LIN {X 0,Y 518.085,Z 283.285,A -85,B 0,C 180,E1 -4909.393,E2 -4909.393} C_VEL
LIN {X 0,Y 517.096,Z 284.359,A -85,B 0,C 180,E1 -4910.032,E2 -4910.032} C_VEL
LIN {X 0,Y 517.024,Z 284.686,A -85,B 0,C 180,E1 -4910.248,E2 -4910.248} C_VEL
LIN {X 0,Y 516.962,Z 289.338,A -85,B 0,C 180,E1 -4913.331,E2 -4913.331} C_VEL
LIN {X 0,Y 516.869,Z 293.688,A -85,B 0,C 180,E1 -4916.119,E2 -4916.119} C_VEL
LIN {X 0,Y 516.72,Z 298.275,A -85,B 0,C 180,E1 -4918.968,E2 -4918.968} C_VEL
LIN {X 0,Y 516.637,Z 302.571,A -85,B 0,C 180,E1 -4921.569,E2 -4921.569} C_VEL
LIN {X 0,Y 516.583,Z 307.01,A -85,B 0,C 180,E1 -4924.193,E2 -4924.193} C_VEL
LIN {X 0,Y 516.487,Z 311.491,A -85,B 0,C 180,E1 -4926.759,E2 -4926.759} C_VEL
LIN {X 0,Y 516.42,Z 317.774,A -85,B 0,C 180,E1 -4930.317,E2 -4930.317} C_VEL
LIN {X 0,Y 516.431,Z 317.992,A -85,B 0,C 180,E1 -4930.439,E2 -4930.439} C_VEL
LIN {X 0,Y 520.62,Z 334.551,A -85,B 0,C 180,E1 -4930.933,E2 -4930.933} C_VEL
LIN {X 0,Y 520.4,Z 349.343,A -85,B 0,C 180,E1 -4931.382,E2 -4931.382} C_VEL
LIN {X 0,Y 519.913,Z 364.135,A -85,B 0,C 180,E1 -4931.989,E2 -4931.989} C_VEL
LIN {X 0,Y 519.41,Z 378.991,A -85,B 0,C 180,E1 -4932.784,E2 -4932.784} C_VEL
LIN {X 0,Y 518.883,Z 392.399,A -85,B 0,C 180,E1 -4933.678,E2 -4933.678} C_VEL
LIN {X 0,Y 518.337,Z 404.939,A -85,B 0,C 180,E1 -4934.694,E2 -4934.694} C_VEL
LIN {X 0,Y 517.847,Z 416.905,A -85,B 0,C 180,E1 -4935.861,E2 -4935.861} C_VEL
LIN {X 0,Y 517.443,Z 427.131,A -85,B 0,C 180,E1 -4937.05,E2 -4937.05} C_VEL
LIN {X 0,Y 517.039,Z 437.144,A -85,B 0,C 180,E1 -4938.435,E2 -4938.435} C_VEL
LIN {X 0,Y 516.76,Z 445.45,A -85,B 0,C 180,E1 -4939.817,E2 -4939.817} C_VEL
LIN {X 0,Y 516.543,Z 453.254,A -85,B 0,C 180,E1 -4941.393,E2 -4941.393} C_VEL
LIN {X 0,Y 516.392,Z 459.47,A -85,B 0,C 180,E1 -4942.965,E2 -4942.965} C_VEL
LIN {X 0,Y 516.374,Z 464.272,A -85,B 0,C 180,E1 -4944.533,E2 -4944.533} C_VEL
LIN {X 0,Y 516.307,Z 467.798,A -85,B 0,C 180,E1 -4946.098,E2 -4946.098} C_VEL
LIN {X 0,Y 516.259,Z 470.138,A -85,B 0,C 180,E1 -4947.66,E2 -4947.66} C_VEL
LIN {X 0,Y 516.156,Z 471.337,A -85,B 0,C 180,E1 -4949.22,E2 -4949.22} C_VEL
LIN {X 0,Y 516.157,Z 471.356,A -85,B 0,C 180,E1 -4950.78,E2 -4950.78} C_VEL
LIN {X 0,Y 516.259,Z 470.234,A -85,B 0,C 180,E1 -4952.341,E2 -4952.341} C_VEL
LIN {X 0,Y 516.308,Z 467.969,A -85,B 0,C 180,E1 -4953.903,E2 -4953.903} C_VEL
LIN {X 0,Y 516.369,Z 464.514,A -85,B 0,C 180,E1 -4955.467,E2 -4955.467} C_VEL
LIN {X 0,Y 516.393,Z 459.789,A -85,B 0,C 180,E1 -4957.036,E2 -4957.036} C_VEL
LIN {X 0,Y 516.541,Z 453.666,A -85,B 0,C 180,E1 -4958.608,E2 -4958.608} C_VEL
LIN {X 0,Y 516.758,Z 445.959,A -85,B 0,C 180,E1 -4960.184,E2 -4960.184} C_VEL
LIN {X 0,Y 516.984,Z 437.741,A -85,B 0,C 180,E1 -4961.567,E2 -4961.567} C_VEL
LIN {X 0,Y 517.4,Z 427.847,A -85,B 0,C 180,E1 -4962.951,E2 -4962.951} C_VEL
LIN {X 0,Y 517.822,Z 417.702,A -85,B 0,C 180,E1 -4964.141,E2 -4964.141} C_VEL
LIN {X 0,Y 518.293,Z 406.094,A -85,B 0,C 180,E1 -4965.289,E2 -4965.289} C_VEL
LIN {X 0,Y 518.821,Z 393.789,A -85,B 0,C 180,E1 -4966.305,E2 -4966.305} C_VEL
LIN {X 0,Y 519.335,Z 380.39,A -85,B 0,C 180,E1 -4967.219,E2 -4967.219} C_VEL
LIN {X 0,Y 519.776,Z 367.881,A -85,B 0,C 180,E1 -4967.915,E2 -4967.915} C_VEL
LIN {X 0,Y 520.298,Z 353.859,A -85,B 0,C 180,E1 -4968.535,E2 -4968.535} C_VEL
LIN {X 0,Y 520.613,Z 339.005,A -85,B 0,C 180,E1 -4969.032,E2 -4969.032} C_VEL
LIN {X 0,Y 520.524,Z 334.046,A -85,B 0,C 180,E1 -4969.173,E2 -4969.173} C_VEL
LIN {X 0,Y 516.438,Z 317.99,A -85,B 0,C 180,E1 -4969.655,E2 -4969.655} C_VEL
LIN {X 0,Y 516.488,Z 311.675,A -85,B 0,C 180,E1 -4973.242,E2 -4973.242} C_VEL
LIN {X 0,Y 516.571,Z 306.704,A -85,B 0,C 180,E1 -4976.112,E2 -4976.112} C_VEL
LIN {X 0,Y 516.696,Z 301.285,A -85,B 0,C 180,E1 -4979.318,E2 -4979.318} C_VEL
LIN {X 0,Y 516.786,Z 296.023,A -85,B 0,C 180,E1 -4982.524,E2 -4982.524} C_VEL
LIN {X 0,Y 516.89,Z 291.549,A -85,B 0,C 180,E1 -4985.333,E2 -4985.333} C_VEL
LIN {X 0,Y 516.975,Z 287.518,A -85,B 0,C 180,E1 -4987.956,E2 -4987.956} C_VEL
LIN {X 0,Y 517.036,Z 283.394,A -85,B 0,C 180,E1 -4990.727,E2 -4990.727} C_VEL
LIN {X 0,Y 516.853,Z 280.732,A -85,B 0,C 180,E1 -4992.754,E2 -4992.754} C_VEL
LIN {X 0,Y 516.922,Z 280.722,A -85,B 0,C 180,E1 -4995.01,E2 -4995.01} C_VEL
LIN {X 0,Y 516.911,Z 280.722,A -85,B 0,C 180,E1 -4998.399,E2 -4998.399} C_VEL
LIN {X 0,Y 516.881,Z 280.725,A -85,B 0,C 180,E1 -5001.284,E2 -5001.284} C_VEL
LIN {X 0,Y 516.865,Z 280.727,A -85,B 0,C 180,E1 -5004.219,E2 -5004.219} C_VEL
LIN {X 0,Y 516.892,Z 280.723,A -85,B 0,C 180,E1 -5007.053,E2 -5007.053} C_VEL
LIN {X 0,Y 516.889,Z 280.725,A -85,B 0,C 180,E1 -5009.796,E2 -5009.796} C_VEL
LIN {X 0,Y 516.894,Z 280.727,A -85,B 0,C 180,E1 -5012.465,E2 -5012.465} C_VEL
LIN {X 0,Y 516.866,Z 280.726,A -85,B 0,C 180,E1 -5015.069,E2 -5015.069} C_VEL
LIN {X 0,Y 516.866,Z 280.725,A -85,B 0,C 180,E1 -5017.621,E2 -5017.621} C_VEL
LIN {X 0,Y 516.928,Z 280.723,A -85,B 0,C 180,E1 -5020.13,E2 -5020.13} C_VEL
LIN {X 0,Y 516.926,Z 280.719,A -85,B 0,C 180,E1 -5022.596,E2 -5022.596} C_VEL
LIN {X 0,Y 516.935,Z 280.72,A -85,B 0,C 180,E1 -5025.03,E2 -5025.03} C_VEL
LIN {X 0,Y 516.962,Z 280.715,A -85,B 0,C 180,E1 -5028.234,E2 -5028.234} C_VEL
LIN {X 0,Y 516.964,Z 280.714,A -85,B 0,C 180,E1 -5031.4,E2 -5031.4} C_VEL
LIN {X 0,Y 517.02,Z 280.707,A -85,B 0,C 180,E1 -5034.54,E2 -5034.54} C_VEL
LIN {X 0,Y 517.082,Z 280.699,A -85,B 0,C 180,E1 -5037.663,E2 -5037.663} C_VEL
LIN {X 0,Y 517.083,Z 280.699,A -85,B 0,C 180,E1 -5040.779,E2 -5040.779} C_VEL
LIN {X 0,Y 517.011,Z 280.712,A -85,B 0,C 180,E1 -5043.117,E2 -5043.117} C_VEL
LIN {X 0,Y 516.983,Z 280.715,A -85,B 0,C 180,E1 -5046.243,E2 -5046.243} C_VEL
LIN {X 0,Y 516.949,Z 280.719,A -85,B 0,C 180,E1 -5049.389,E2 -5049.389} C_VEL
LIN {X 0,Y 516.948,Z 280.717,A -85,B 0,C 180,E1 -5051.807,E2 -5051.807} C_VEL
LIN {X 0,Y 516.939,Z 280.72,A -85,B 0,C 180,E1 -5055.146,E2 -5055.146} C_VEL
LIN {X 0,Y 516.921,Z 280.722,A -85,B 0,C 180,E1 -5058.222,E2 -5058.222} C_VEL
LIN {X 0,Y 516.9,Z 280.721,A -85,B 0,C 180,E1 -5060.702,E2 -5060.702} C_VEL
LIN {X 0,Y 516.899,Z 280.723,A -85,B 0,C 180,E1 -5064.072,E2 -5064.072} C_VEL
LIN {X 0,Y 516.918,Z 280.72,A -85,B 0,C 180,E1 -5066.658,E2 -5066.658} C_VEL
LIN {X 0,Y 516.904,Z 280.724,A -85,B 0,C 180,E1 -5069.523,E2 -5069.523} C_VEL
LIN {X 0,Y 516.892,Z 280.726,A -85,B 0,C 180,E1 -5072.544,E2 -5072.544} C_VEL
LIN {X 0,Y 516.859,Z 280.734,A -85,B 0,C 180,E1 -5075.329,E2 -5075.329} C_VEL
LIN {X 0,Y 516.879,Z 280.729,A -85,B 0,C 180,E1 -5077.943,E2 -5077.943} C_VEL
LIN {X 0,Y 516.879,Z 280.726,A -85,B 0,C 180,E1 -5080.742,E2 -5080.742} C_VEL
LIN {X 0,Y 516.879,Z 280.728,A -85,B 0,C 180,E1 -5083.903,E2 -5083.903} C_VEL
LIN {X 0,Y 516.957,Z 280.907,A -85,B 0,C 180,E1 -5086.643,E2 -5086.643} C_VEL
LIN {X 0,Y 517.284,Z 283.704,A -85,B 0,C 180,E1 -5088.352,E2 -5088.352} C_VEL
LIN {X 0,Y 517.265,Z 287.849,A -85,B 0,C 180,E1 -5090.755,E2 -5090.755} C_VEL
LIN {X 0,Y 517.156,Z 292.427,A -85,B 0,C 180,E1 -5093.301,E2 -5093.301} C_VEL
LIN {X 0,Y 517.023,Z 297.711,A -85,B 0,C 180,E1 -5096.13,E2 -5096.13} C_VEL
LIN {X 0,Y 516.879,Z 303.124,A -85,B 0,C 180,E1 -5098.938,E2 -5098.938} C_VEL
LIN {X 0,Y 516.74,Z 308.364,A -85,B 0,C 180,E1 -5101.574,E2 -5101.574} C_VEL
LIN {X 0,Y 516.639,Z 313.709,A -85,B 0,C 180,E1 -5104.195,E2 -5104.195} C_VEL
LIN {X 0,Y 516.54,Z 319.079,A -85,B 0,C 180,E1 -5106.761,E2 -5106.761} C_VEL
LIN {X 0,Y 516.501,Z 325.688,A -85,B 0,C 180,E1 -5109.864,E2 -5109.864} C_VEL
LIN {X 0,Y 516.49,Z 326.814,A -85,B 0,C 180,E1 -5110.387,E2 -5110.387} C_VEL
LIN {X 0,Y 520.37,Z 342.561,A -85,B 0,C 180,E1 -5110.842,E2 -5110.842} C_VEL
LIN {X 0,Y 520.646,Z 345.506,A -85,B 0,C 180,E1 -5110.929,E2 -5110.929} C_VEL
LIN {X 0,Y 520.355,Z 359.33,A -85,B 0,C 180,E1 -5111.351,E2 -5111.351} C_VEL
LIN {X 0,Y 519.86,Z 373.609,A -85,B 0,C 180,E1 -5111.935,E2 -5111.935} C_VEL
LIN {X 0,Y 519.383,Z 387.714,A -85,B 0,C 180,E1 -5112.681,E2 -5112.681} C_VEL
LIN {X 0,Y 518.869,Z 401.448,A -85,B 0,C 180,E1 -5113.586,E2 -5113.586} C_VEL
LIN {X 0,Y 518.368,Z 413.415,A -85,B 0,C 180,E1 -5114.542,E2 -5114.542} C_VEL
LIN {X 0,Y 517.873,Z 425.158,A -85,B 0,C 180,E1 -5115.66,E2 -5115.66} C_VEL
LIN {X 0,Y 517.466,Z 435.667,A -85,B 0,C 180,E1 -5116.85,E2 -5116.85} C_VEL
LIN {X 0,Y 517.013,Z 445.939,A -85,B 0,C 180,E1 -5118.235,E2 -5118.235} C_VEL
LIN {X 0,Y 516.833,Z 454.478,A -85,B 0,C 180,E1 -5119.62,E2 -5119.62} C_VEL
LIN {X 0,Y 516.588,Z 461.58,A -85,B 0,C 180,E1 -5120.999,E2 -5120.999} C_VEL
LIN {X 0,Y 516.429,Z 468.166,A -85,B 0,C 180,E1 -5122.572,E2 -5122.572} C_VEL
LIN {X 0,Y 516.378,Z 473.318,A -85,B 0,C 180,E1 -5124.141,E2 -5124.141} C_VEL
LIN {X 0,Y 516.239,Z 476.289,A -85,B 0,C 180,E1 -5125.314,E2 -5125.314} C_VEL
LIN {X 0,Y 516.271,Z 479.183,A -85,B 0,C 180,E1 -5126.878,E2 -5126.878} C_VEL
LIN {X 0,Y 516.189,Z 480.908,A -85,B 0,C 180,E1 -5128.439,E2 -5128.439} C_VEL
LIN {X 0,Y 516.151,Z 481.5,A -85,B 0,C 180,E1 -5130,E2 -5130} C_VEL
LIN {X 0,Y 516.189,Z 480.906,A -85,B 0,C 180,E1 -5131.56,E2 -5131.56} C_VEL
LIN {X 0,Y 516.271,Z 479.178,A -85,B 0,C 180,E1 -5133.121,E2 -5133.121} C_VEL
LIN {X 0,Y 516.239,Z 476.288,A -85,B 0,C 180,E1 -5134.685,E2 -5134.685} C_VEL
LIN {X 0,Y 516.375,Z 472.162,A -85,B 0,C 180,E1 -5136.25,E2 -5136.25} C_VEL
LIN {X 0,Y 516.462,Z 466.681,A -85,B 0,C 180,E1 -5137.821,E2 -5137.821} C_VEL
LIN {X 0,Y 516.637,Z 459.705,A -85,B 0,C 180,E1 -5139.395,E2 -5139.395} C_VEL
LIN {X 0,Y 516.952,Z 451.021,A -85,B 0,C 180,E1 -5140.972,E2 -5140.972} C_VEL
LIN {X 0,Y 517.225,Z 441.942,A -85,B 0,C 180,E1 -5142.337,E2 -5142.337} C_VEL
LIN {X 0,Y 517.607,Z 432.409,A -85,B 0,C 180,E1 -5143.545,E2 -5143.545} C_VEL
LIN {X 0,Y 518.096,Z 420.241,A -85,B 0,C 180,E1 -5144.835,E2 -5144.835} C_VEL
LIN {X 0,Y 518.62,Z 408.084,A -85,B 0,C 180,E1 -5145.906,E2 -5145.906} C_VEL
LIN {X 0,Y 519.074,Z 395.608,A -85,B 0,C 180,E1 -5146.822,E2 -5146.822} C_VEL
LIN {X 0,Y 519.562,Z 382.415,A -85,B 0,C 180,E1 -5147.617,E2 -5147.617} C_VEL
LIN {X 0,Y 520.124,Z 367.924,A -85,B 0,C 180,E1 -5148.312,E2 -5148.312} C_VEL
LIN {X 0,Y 520.484,Z 353.145,A -85,B 0,C 180,E1 -5148.855,E2 -5148.855} C_VEL
LIN {X 0,Y 520.53,Z 343.102,A -85,B 0,C 180,E1 -5149.14,E2 -5149.14} C_VEL
LIN {X 0,Y 516.483,Z 326.786,A -85,B 0,C 180,E1 -5149.633,E2 -5149.633} C_VEL
LIN {X 0,Y 516.53,Z 320.903,A -85,B 0,C 180,E1 -5152.393,E2 -5152.393} C_VEL
LIN {X 0,Y 516.597,Z 315.556,A -85,B 0,C 180,E1 -5154.944,E2 -5154.944} C_VEL
LIN {X 0,Y 516.713,Z 309.555,A -85,B 0,C 180,E1 -5157.861,E2 -5157.861} C_VEL
LIN {X 0,Y 516.832,Z 304.84,A -85,B 0,C 180,E1 -5160.207,E2 -5160.207} C_VEL
LIN {X 0,Y 516.947,Z 299.493,A -85,B 0,C 180,E1 -5162.942,E2 -5162.942} C_VEL
LIN {X 0,Y 517.096,Z 294.159,A -85,B 0,C 180,E1 -5165.761,E2 -5165.761} C_VEL
LIN {X 0,Y 517.254,Z 288.849,A -85,B 0,C 180,E1 -5168.682,E2 -5168.682} C_VEL
LIN {X 0,Y 517.343,Z 285.301,A -85,B 0,C 180,E1 -5170.697,E2 -5170.697} C_VEL
LIN {X 0,Y 517.061,Z 281.779,A -85,B 0,C 180,E1 -5172.812,E2 -5172.812} C_VEL
LIN {X 0,Y 516.918,Z 280.722,A -85,B 0,C 180,E1 -5173.515,E2 -5173.515} C_VEL
LIN {X 0,Y 516.876,Z 280.728,A -85,B 0,C 180,E1 -5176.106,E2 -5176.106} C_VEL
LIN {X 0,Y 516.908,Z 280.725,A -85,B 0,C 180,E1 -5178.398,E2 -5178.398} C_VEL
LIN {X 0,Y 516.877,Z 280.726,A -85,B 0,C 180,E1 -5181.284,E2 -5181.284} C_VEL
LIN {X 0,Y 516.86,Z 280.728,A -85,B 0,C 180,E1 -5184.219,E2 -5184.219} C_VEL
LIN {X 0,Y 516.89,Z 280.725,A -85,B 0,C 180,E1 -5187.053,E2 -5187.053} C_VEL
LIN {X 0,Y 516.884,Z 280.727,A -85,B 0,C 180,E1 -5189.796,E2 -5189.796} C_VEL
LIN {X 0,Y 516.914,Z 280.725,A -85,B 0,C 180,E1 -5192.467,E2 -5192.467} C_VEL
LIN {X 0,Y 516.903,Z 280.722,A -85,B 0,C 180,E1 -5195.072,E2 -5195.072} C_VEL
LIN {X 0,Y 516.861,Z 280.727,A -85,B 0,C 180,E1 -5197.621,E2 -5197.621} C_VEL
LIN {X 0,Y 516.924,Z 280.723,A -85,B 0,C 180,E1 -5200.13,E2 -5200.13} C_VEL
LIN {X 0,Y 516.92,Z 280.719,A -85,B 0,C 180,E1 -5202.596,E2 -5202.596} C_VEL
LIN {X 0,Y 516.931,Z 280.719,A -85,B 0,C 180,E1 -5205.03,E2 -5205.03} C_VEL
LIN {X 0,Y 516.956,Z 280.715,A -85,B 0,C 180,E1 -5208.234,E2 -5208.234} C_VEL
LIN {X 0,Y 516.96,Z 280.714,A -85,B 0,C 180,E1 -5211.4,E2 -5211.4} C_VEL
LIN {X 0,Y 517.017,Z 280.706,A -85,B 0,C 180,E1 -5214.54,E2 -5214.54} C_VEL
LIN {X 0,Y 517.079,Z 280.697,A -85,B 0,C 180,E1 -5217.663,E2 -5217.663} C_VEL
LIN {X 0,Y 517.08,Z 280.699,A -85,B 0,C 180,E1 -5220.779,E2 -5220.779} C_VEL
LIN {X 0,Y 517.009,Z 280.713,A -85,B 0,C 180,E1 -5223.117,E2 -5223.117} C_VEL
LIN {X 0,Y 516.979,Z 280.716,A -85,B 0,C 180,E1 -5226.244,E2 -5226.244} C_VEL
LIN {X 0,Y 516.946,Z 280.719,A -85,B 0,C 180,E1 -5229.389,E2 -5229.389} C_VEL
LIN {X 0,Y 516.943,Z 280.716,A -85,B 0,C 180,E1 -5231.807,E2 -5231.807} C_VEL
LIN {X 0,Y 516.934,Z 280.72,A -85,B 0,C 180,E1 -5235.146,E2 -5235.146} C_VEL
LIN {X 0,Y 516.918,Z 280.722,A -85,B 0,C 180,E1 -5238.223,E2 -5238.223} C_VEL
LIN {X 0,Y 516.904,Z 280.72,A -85,B 0,C 180,E1 -5240.702,E2 -5240.702} C_VEL
LIN {X 0,Y 516.904,Z 280.722,A -85,B 0,C 180,E1 -5244.072,E2 -5244.072} C_VEL
LIN {X 0,Y 516.915,Z 280.719,A -85,B 0,C 180,E1 -5246.658,E2 -5246.658} C_VEL
LIN {X 0,Y 516.903,Z 280.721,A -85,B 0,C 180,E1 -5249.524,E2 -5249.524} C_VEL
LIN {X 0,Y 516.894,Z 280.722,A -85,B 0,C 180,E1 -5252.545,E2 -5252.545} C_VEL
LIN {X 0,Y 516.856,Z 280.73,A -85,B 0,C 180,E1 -5255.33,E2 -5255.33} C_VEL
LIN {X 0,Y 516.876,Z 280.727,A -85,B 0,C 180,E1 -5257.944,E2 -5257.944} C_VEL
LIN {X 0,Y 516.879,Z 280.725,A -85,B 0,C 180,E1 -5260.742,E2 -5260.742} C_VEL
LIN {X 0,Y 516.877,Z 280.73,A -85,B 0,C 180,E1 -5262.832,E2 -5262.832} C_VEL
LIN {X 0,Y 516.918,Z 280.72,A -85,B 0,C 180,E1 -5265.011,E2 -5265.011} C_VEL
LIN {X 0,Y 516.851,Z 280.732,A -85,B 0,C 180,E1 -5267.246,E2 -5267.246} C_VEL
LIN {X 0,Y 516.99,Z 281.991,A -85,B 0,C 180,E1 -5268.389,E2 -5268.389} C_VEL
LIN {X 0,Y 517.024,Z 284.686,A -85,B 0,C 180,E1 -5270.248,E2 -5270.248} C_VEL
LIN {X 0,Y 516.373,Z 285.721,A -85,B 0,C 180,E1 -5270.888,E2 -5270.888} C_VEL
LIN {X 0,Y 513.494,Z 287.66,A -85,B 0,C 180,E1 -5271.92,E2 -5271.92} C_VEL
LIN {X 0,Y 511.04,Z 289.243,A -85,B 0,C 180,E1 -5272.751,E2 -5272.751} C_VEL
LIN {X 0,Y 509.979,Z 290.355,A -85,B 0,C 180,E1 -5273.395,E2 -5273.395} C_VEL
LIN {X 0,Y 509.89,Z 290.698,A -85,B 0,C 180,E1 -5273.614,E2 -5273.614} C_VEL
LIN {X 0,Y 509.782,Z 295.211,A -85,B 0,C 180,E1 -5276.534,E2 -5276.534} C_VEL
LIN {X 0,Y 509.645,Z 299.658,A -85,B 0,C 180,E1 -5279.322,E2 -5279.322} C_VEL
LIN {X 0,Y 509.591,Z 304.098,A -85,B 0,C 180,E1 -5282.037,E2 -5282.037} C_VEL
LIN {X 0,Y 509.485,Z 308.546,A -85,B 0,C 180,E1 -5284.684,E2 -5284.684} C_VEL
LIN {X 0,Y 509.378,Z 313.561,A -85,B 0,C 180,E1 -5287.58,E2 -5287.58} C_VEL
LIN {X 0,Y 509.369,Z 318.129,A -85,B 0,C 180,E1 -5290.159,E2 -5290.159} C_VEL
LIN {X 0,Y 513.592,Z 334.488,A -85,B 0,C 180,E1 -5290.658,E2 -5290.658} C_VEL
LIN {X 0,Y 513.933,Z 338.016,A -85,B 0,C 180,E1 -5290.771,E2 -5290.771} C_VEL
LIN {X 0,Y 513.555,Z 353.574,A -85,B 0,C 180,E1 -5291.289,E2 -5291.289} C_VEL
LIN {X 0,Y 512.971,Z 368.2,A -85,B 0,C 180,E1 -5291.943,E2 -5291.943} C_VEL
LIN {X 0,Y 512.443,Z 382.231,A -85,B 0,C 180,E1 -5292.748,E2 -5292.748} C_VEL
LIN {X 0,Y 511.923,Z 395.059,A -85,B 0,C 180,E1 -5293.655,E2 -5293.655} C_VEL
LIN {X 0,Y 511.331,Z 407.169,A -85,B 0,C 180,E1 -5294.684,E2 -5294.684} C_VEL
LIN {X 0,Y 510.83,Z 418.764,A -85,B 0,C 180,E1 -5295.866,E2 -5295.866} C_VEL
LIN {X 0,Y 510.39,Z 428.745,A -85,B 0,C 180,E1 -5297.071,E2 -5297.071} C_VEL
LIN {X 0,Y 510,Z 438.702,A -85,B 0,C 180,E1 -5298.508,E2 -5298.508} C_VEL
LIN {X 0,Y 509.7,Z 446.621,A -85,B 0,C 180,E1 -5299.875,E2 -5299.875} C_VEL
LIN {X 0,Y 509.487,Z 453.326,A -85,B 0,C 180,E1 -5301.273,E2 -5301.273} C_VEL
LIN {X 0,Y 509.319,Z 459.541,A -85,B 0,C 180,E1 -5302.866,E2 -5302.866} C_VEL
LIN {X 0,Y 509.305,Z 464.343,A -85,B 0,C 180,E1 -5304.457,E2 -5304.457} C_VEL
LIN {X 0,Y 509.202,Z 467.865,A -85,B 0,C 180,E1 -5306.043,E2 -5306.043} C_VEL
LIN {X 0,Y 509.187,Z 470.197,A -85,B 0,C 180,E1 -5307.627,E2 -5307.627} C_VEL
LIN {X 0,Y 509.07,Z 471.393,A -85,B 0,C 180,E1 -5309.209,E2 -5309.209} C_VEL
LIN {X 0,Y 509.071,Z 471.412,A -85,B 0,C 180,E1 -5310.791,E2 -5310.791} C_VEL
LIN {X 0,Y 509.188,Z 470.291,A -85,B 0,C 180,E1 -5312.373,E2 -5312.373} C_VEL
LIN {X 0,Y 509.202,Z 468.033,A -85,B 0,C 180,E1 -5313.957,E2 -5313.957} C_VEL
LIN {X 0,Y 509.299,Z 464.581,A -85,B 0,C 180,E1 -5315.543,E2 -5315.543} C_VEL
LIN {X 0,Y 509.319,Z 459.856,A -85,B 0,C 180,E1 -5317.134,E2 -5317.134} C_VEL
LIN {X 0,Y 509.485,Z 453.733,A -85,B 0,C 180,E1 -5318.728,E2 -5318.728} C_VEL
LIN {X 0,Y 509.747,Z 446.025,A -85,B 0,C 180,E1 -5320.325,E2 -5320.325} C_VEL
LIN {X 0,Y 510.01,Z 437.485,A -85,B 0,C 180,E1 -5321.777,E2 -5321.777} C_VEL
LIN {X 0,Y 510.415,Z 427.912,A -85,B 0,C 180,E1 -5323.132,E2 -5323.132} C_VEL
LIN {X 0,Y 510.879,Z 417.766,A -85,B 0,C 180,E1 -5324.337,E2 -5324.337} C_VEL
LIN {X 0,Y 511.394,Z 406.478,A -85,B 0,C 180,E1 -5325.469,E2 -5325.469} C_VEL
LIN {X 0,Y 511.987,Z 393.592,A -85,B 0,C 180,E1 -5326.549,E2 -5326.549} C_VEL
LIN {X 0,Y 512.545,Z 380.449,A -85,B 0,C 180,E1 -5327.455,E2 -5327.455} C_VEL
LIN {X 0,Y 513.008,Z 367.937,A -85,B 0,C 180,E1 -5328.16,E2 -5328.16} C_VEL
LIN {X 0,Y 513.55,Z 354.34,A -85,B 0,C 180,E1 -5328.77,E2 -5328.77} C_VEL
LIN {X 0,Y 513.89,Z 339.691,A -85,B 0,C 180,E1 -5329.273,E2 -5329.273} C_VEL
LIN {X 0,Y 513.789,Z 335.166,A -85,B 0,C 180,E1 -5329.405,E2 -5329.405} C_VEL
LIN {X 0,Y 509.755,Z 320.075,A -85,B 0,C 180,E1 -5329.883,E2 -5329.883} C_VEL
LIN {X 0,Y 509.368,Z 318.036,A -85,B 0,C 180,E1 -5329.955,E2 -5329.955} C_VEL
LIN {X 0,Y 509.419,Z 311.73,A -85,B 0,C 180,E1 -5333.584,E2 -5333.584} C_VEL
LIN {X 0,Y 509.505,Z 307.119,A -85,B 0,C 180,E1 -5336.286,E2 -5336.286} C_VEL
LIN {X 0,Y 509.596,Z 302.818,A -85,B 0,C 180,E1 -5338.861,E2 -5338.861} C_VEL
LIN {X 0,Y 509.679,Z 298.356,A -85,B 0,C 180,E1 -5341.6,E2 -5341.6} C_VEL
LIN {X 0,Y 509.837,Z 293.877,A -85,B 0,C 180,E1 -5344.414,E2 -5344.414} C_VEL
LIN {X 0,Y 509.945,Z 289.406,A -85,B 0,C 180,E1 -5347.329,E2 -5347.329} C_VEL
LIN {X 0,Y 510.016,Z 284.924,A -85,B 0,C 180,E1 -5350.365,E2 -5350.365} C_VEL
LIN {X 0,Y 509.843,Z 281.923,A -85,B 0,C 180,E1 -5352.488,E2 -5352.488} C_VEL
LIN {X 0,Y 509.808,Z 281.608,A -85,B 0,C 180,E1 -5353.573,E2 -5353.573} C_VEL
LIN {X 0,Y 509.817,Z 281.606,A -85,B 0,C 180,E1 -5356.428,E2 -5356.428} C_VEL
LIN {X 0,Y 509.836,Z 281.602,A -85,B 0,C 180,E1 -5359.302,E2 -5359.302} C_VEL
LIN {X 0,Y 509.85,Z 281.606,A -85,B 0,C 180,E1 -5361.786,E2 -5361.786} C_VEL
LIN {X 0,Y 509.824,Z 281.607,A -85,B 0,C 180,E1 -5364.621,E2 -5364.621} C_VEL
LIN {X 0,Y 509.859,Z 281.6,A -85,B 0,C 180,E1 -5367.481,E2 -5367.481} C_VEL
LIN {X 0,Y 509.856,Z 281.599,A -85,B 0,C 180,E1 -5370.273,E2 -5370.273} C_VEL
LIN {X 0,Y 509.876,Z 281.597,A -85,B 0,C 180,E1 -5373.629,E2 -5373.629} C_VEL
LIN {X 0,Y 509.827,Z 281.603,A -85,B 0,C 180,E1 -5376.436,E2 -5376.436} C_VEL
LIN {X 0,Y 509.911,Z 281.594,A -85,B 0,C 180,E1 -5379.844,E2 -5379.844} C_VEL
LIN {X 0,Y 509.88,Z 281.6,A -85,B 0,C 180,E1 -5383.175,E2 -5383.175} C_VEL
LIN {X 0,Y 509.851,Z 281.6,A -85,B 0,C 180,E1 -5385.634,E2 -5385.634} C_VEL
LIN {X 0,Y 509.91,Z 281.593,A -85,B 0,C 180,E1 -5388.874,E2 -5388.874} C_VEL
LIN {X 0,Y 509.916,Z 281.593,A -85,B 0,C 180,E1 -5392.078,E2 -5392.078} C_VEL
LIN {X 0,Y 509.97,Z 281.585,A -85,B 0,C 180,E1 -5394.464,E2 -5394.464} C_VEL
LIN {X 0,Y 510.053,Z 281.574,A -85,B 0,C 180,E1 -5397.631,E2 -5397.631} C_VEL
LIN {X 0,Y 510.052,Z 281.579,A -85,B 0,C 180,E1 -5400,E2 -5400} C_VEL
LIN {X 0,Y 510.053,Z 281.575,A -85,B 0,C 180,E1 -5402.369,E2 -5402.369} C_VEL
LIN {X 0,Y 509.971,Z 281.585,A -85,B 0,C 180,E1 -5405.536,E2 -5405.536} C_VEL
LIN {X 0,Y 509.91,Z 281.593,A -85,B 0,C 180,E1 -5408.72,E2 -5408.72} C_VEL
LIN {X 0,Y 509.9,Z 281.595,A -85,B 0,C 180,E1 -5411.932,E2 -5411.932} C_VEL
LIN {X 0,Y 509.89,Z 281.599,A -85,B 0,C 180,E1 -5415.242,E2 -5415.242} C_VEL
LIN {X 0,Y 509.885,Z 281.597,A -85,B 0,C 180,E1 -5418.001,E2 -5418.001} C_VEL
LIN {X 0,Y 509.842,Z 281.602,A -85,B 0,C 180,E1 -5421.002,E2 -5421.002} C_VEL
LIN {X 0,Y 509.861,Z 281.603,A -85,B 0,C 180,E1 -5424.426,E2 -5424.426} C_VEL
LIN {X 0,Y 509.877,Z 281.598,A -85,B 0,C 180,E1 -5427.056,E2 -5427.056} C_VEL
LIN {X 0,Y 509.853,Z 281.601,A -85,B 0,C 180,E1 -5429.751,E2 -5429.751} C_VEL
LIN {X 0,Y 509.87,Z 281.6,A -85,B 0,C 180,E1 -5432.774,E2 -5432.774} C_VEL
LIN {X 0,Y 509.819,Z 281.608,A -85,B 0,C 180,E1 -5435.578,E2 -5435.578} C_VEL
LIN {X 0,Y 509.848,Z 281.607,A -85,B 0,C 180,E1 -5438.338,E2 -5438.338} C_VEL
LIN {X 0,Y 509.849,Z 281.605,A -85,B 0,C 180,E1 -5441.426,E2 -5441.426} C_VEL
LIN {X 0,Y 509.855,Z 281.606,A -85,B 0,C 180,E1 -5444.668,E2 -5444.668} C_VEL
LIN {X 0,Y 509.884,Z 281.764,A -85,B 0,C 180,E1 -5446.436,E2 -5446.436} C_VEL
LIN {X 0,Y 510.297,Z 285.291,A -85,B 0,C 180,E1 -5448.619,E2 -5448.619} C_VEL
LIN {X 0,Y 510.247,Z 288.818,A -85,B 0,C 180,E1 -5450.685,E2 -5450.685} C_VEL
LIN {X 0,Y 510.113,Z 294.124,A -85,B 0,C 180,E1 -5453.671,E2 -5453.671} C_VEL
LIN {X 0,Y 509.94,Z 299.443,A -85,B 0,C 180,E1 -5456.545,E2 -5456.545} C_VEL
LIN {X 0,Y 509.812,Z 304.758,A -85,B 0,C 180,E1 -5459.332,E2 -5459.332} C_VEL
LIN {X 0,Y 509.657,Z 310.091,A -85,B 0,C 180,E1 -5462.041,E2 -5462.041} C_VEL
LIN {X 0,Y 509.535,Z 315.431,A -85,B 0,C 180,E1 -5464.686,E2 -5464.686} C_VEL
LIN {X 0,Y 509.458,Z 321.376,A -85,B 0,C 180,E1 -5467.558,E2 -5467.558} C_VEL
LIN {X 0,Y 509.409,Z 326.722,A -85,B 0,C 180,E1 -5470.094,E2 -5470.094} C_VEL
LIN {X 0,Y 513.775,Z 344.464,A -85,B 0,C 180,E1 -5470.636,E2 -5470.636} C_VEL
LIN {X 0,Y 513.603,Z 359.417,A -85,B 0,C 180,E1 -5471.103,E2 -5471.103} C_VEL
LIN {X 0,Y 513.095,Z 373.54,A -85,B 0,C 180,E1 -5471.689,E2 -5471.689} C_VEL
LIN {X 0,Y 512.57,Z 387.645,A -85,B 0,C 180,E1 -5472.443,E2 -5472.443} C_VEL
LIN {X 0,Y 512.019,Z 401.238,A -85,B 0,C 180,E1 -5473.35,E2 -5473.35} C_VEL
LIN {X 0,Y 511.451,Z 413.94,A -85,B 0,C 180,E1 -5474.38,E2 -5474.38} C_VEL
LIN {X 0,Y 510.942,Z 425.088,A -85,B 0,C 180,E1 -5475.462,E2 -5475.462} C_VEL
LIN {X 0,Y 510.487,Z 435.598,A -85,B 0,C 180,E1 -5476.667,E2 -5476.667} C_VEL
LIN {X 0,Y 510.09,Z 444.513,A -85,B 0,C 180,E1 -5477.871,E2 -5477.871} C_VEL
LIN {X 0,Y 509.83,Z 453.289,A -85,B 0,C 180,E1 -5479.275,E2 -5479.275} C_VEL
LIN {X 0,Y 509.556,Z 459.639,A -85,B 0,C 180,E1 -5480.473,E2 -5480.473} C_VEL
LIN {X 0,Y 509.385,Z 466.609,A -85,B 0,C 180,E1 -5482.069,E2 -5482.069} C_VEL
LIN {X 0,Y 509.266,Z 472.087,A -85,B 0,C 180,E1 -5483.661,E2 -5483.661} C_VEL
LIN {X 0,Y 509.159,Z 476.227,A -85,B 0,C 180,E1 -5485.249,E2 -5485.249} C_VEL
LIN {X 0,Y 509.188,Z 479.13,A -85,B 0,C 180,E1 -5486.835,E2 -5486.835} C_VEL
LIN {X 0,Y 509.11,Z 480.861,A -85,B 0,C 180,E1 -5488.418,E2 -5488.418} C_VEL
LIN {X 0,Y 509.062,Z 481.454,A -85,B 0,C 180,E1 -5490,E2 -5490} C_VEL
LIN {X 0,Y 509.11,Z 480.859,A -85,B 0,C 180,E1 -5491.582,E2 -5491.582} C_VEL
LIN {X 0,Y 509.188,Z 479.126,A -85,B 0,C 180,E1 -5493.165,E2 -5493.165} C_VEL
LIN {X 0,Y 509.159,Z 476.226,A -85,B 0,C 180,E1 -5494.75,E2 -5494.75} C_VEL
LIN {X 0,Y 509.305,Z 472.093,A -85,B 0,C 180,E1 -5496.338,E2 -5496.338} C_VEL
LIN {X 0,Y 509.384,Z 466.612,A -85,B 0,C 180,E1 -5497.93,E2 -5497.93} C_VEL
LIN {X 0,Y 509.555,Z 459.635,A -85,B 0,C 180,E1 -5499.526,E2 -5499.526} C_VEL
LIN {X 0,Y 509.882,Z 452.168,A -85,B 0,C 180,E1 -5500.925,E2 -5500.925} C_VEL
LIN {X 0,Y 510.143,Z 443.433,A -85,B 0,C 180,E1 -5502.289,E2 -5502.289} C_VEL
LIN {X 0,Y 510.584,Z 433.972,A -85,B 0,C 180,E1 -5503.532,E2 -5503.532} C_VEL
LIN {X 0,Y 511.034,Z 423.143,A -85,B 0,C 180,E1 -5504.739,E2 -5504.739} C_VEL
LIN {X 0,Y 511.569,Z 411.474,A -85,B 0,C 180,E1 -5505.832,E2 -5505.832} C_VEL
LIN {X 0,Y 512.089,Z 398.395,A -85,B 0,C 180,E1 -5506.853,E2 -5506.853} C_VEL
LIN {X 0,Y 512.695,Z 384.113,A -85,B 0,C 180,E1 -5507.758,E2 -5507.758} C_VEL
LIN {X 0,Y 513.315,Z 369.506,A -85,B 0,C 180,E1 -5508.488,E2 -5508.488} C_VEL
LIN {X 0,Y 513.726,Z 354.274,A -85,B 0,C 180,E1 -5509.071,E2 -5509.071} C_VEL
LIN {X 0,Y 513.79,Z 344.288,A -85,B 0,C 180,E1 -5509.369,E2 -5509.369} C_VEL
LIN {X 0,Y 509.617,Z 328.121,A -85,B 0,C 180,E1 -5509.866,E2 -5509.866} C_VEL
LIN {X 0,Y 509.407,Z 326.717,A -85,B 0,C 180,E1 -5509.915,E2 -5509.915} C_VEL
LIN {X 0,Y 509.448,Z 320.829,A -85,B 0,C 180,E1 -5512.722,E2 -5512.722} C_VEL
LIN {X 0,Y 509.535,Z 315.492,A -85,B 0,C 180,E1 -5515.313,E2 -5515.313} C_VEL
LIN {X 0,Y 509.663,Z 309.964,A -85,B 0,C 180,E1 -5518.051,E2 -5518.051} C_VEL
LIN {X 0,Y 509.813,Z 304.797,A -85,B 0,C 180,E1 -5520.667,E2 -5520.667} C_VEL
LIN {X 0,Y 509.937,Z 299.451,A -85,B 0,C 180,E1 -5523.454,E2 -5523.454} C_VEL
LIN {X 0,Y 510.109,Z 294.121,A -85,B 0,C 180,E1 -5526.329,E2 -5526.329} C_VEL
LIN {X 0,Y 510.253,Z 288.437,A -85,B 0,C 180,E1 -5529.528,E2 -5529.528} C_VEL
LIN {X 0,Y 510.294,Z 285.28,A -85,B 0,C 180,E1 -5531.381,E2 -5531.381} C_VEL
LIN {X 0,Y 509.858,Z 281.599,A -85,B 0,C 180,E1 -5533.694,E2 -5533.694} C_VEL
LIN {X 0,Y 509.812,Z 281.607,A -85,B 0,C 180,E1 -5536.428,E2 -5536.428} C_VEL
LIN {X 0,Y 509.833,Z 281.603,A -85,B 0,C 180,E1 -5539.302,E2 -5539.302} C_VEL
LIN {X 0,Y 509.845,Z 281.606,A -85,B 0,C 180,E1 -5541.786,E2 -5541.786} C_VEL
LIN {X 0,Y 509.819,Z 281.609,A -85,B 0,C 180,E1 -5544.621,E2 -5544.621} C_VEL
LIN {X 0,Y 509.858,Z 281.603,A -85,B 0,C 180,E1 -5547.481,E2 -5547.481} C_VEL
LIN {X 0,Y 509.85,Z 281.602,A -85,B 0,C 180,E1 -5550.273,E2 -5550.273} C_VEL
LIN {X 0,Y 509.873,Z 281.599,A -85,B 0,C 180,E1 -5552.944,E2 -5552.944} C_VEL
LIN {X 0,Y 509.862,Z 281.603,A -85,B 0,C 180,E1 -5555.574,E2 -5555.574} C_VEL
LIN {X 0,Y 509.841,Z 281.602,A -85,B 0,C 180,E1 -5558.998,E2 -5558.998} C_VEL
LIN {X 0,Y 509.88,Z 281.597,A -85,B 0,C 180,E1 -5561.999,E2 -5561.999} C_VEL
LIN {X 0,Y 509.902,Z 281.596,A -85,B 0,C 180,E1 -5564.819,E2 -5564.819} C_VEL
LIN {X 0,Y 509.896,Z 281.595,A -85,B 0,C 180,E1 -5568.121,E2 -5568.121} C_VEL
LIN {X 0,Y 509.907,Z 281.593,A -85,B 0,C 180,E1 -5571.28,E2 -5571.28} C_VEL
LIN {X 0,Y 509.967,Z 281.584,A -85,B 0,C 180,E1 -5574.464,E2 -5574.464} C_VEL
LIN {X 0,Y 510.049,Z 281.573,A -85,B 0,C 180,E1 -5577.631,E2 -5577.631} C_VEL
LIN {X 0,Y 510.051,Z 281.575,A -85,B 0,C 180,E1 -5580.79,E2 -5580.79} C_VEL
LIN {X 0,Y 509.951,Z 281.591,A -85,B 0,C 180,E1 -5583.16,E2 -5583.16} C_VEL
LIN {X 0,Y 509.925,Z 281.593,A -85,B 0,C 180,E1 -5586.33,E2 -5586.33} C_VEL
LIN {X 0,Y 509.906,Z 281.592,A -85,B 0,C 180,E1 -5588.72,E2 -5588.72} C_VEL
LIN {X 0,Y 509.895,Z 281.595,A -85,B 0,C 180,E1 -5591.932,E2 -5591.932} C_VEL
LIN {X 0,Y 509.885,Z 281.599,A -85,B 0,C 180,E1 -5595.242,E2 -5595.242} C_VEL
LIN {X 0,Y 509.881,Z 281.596,A -85,B 0,C 180,E1 -5598.001,E2 -5598.001} C_VEL
LIN {X 0,Y 509.842,Z 281.601,A -85,B 0,C 180,E1 -5601.002,E2 -5601.002} C_VEL
LIN {X 0,Y 509.862,Z 281.603,A -85,B 0,C 180,E1 -5604.426,E2 -5604.426} C_VEL
LIN {X 0,Y 509.874,Z 281.597,A -85,B 0,C 180,E1 -5607.056,E2 -5607.056} C_VEL
LIN {X 0,Y 509.85,Z 281.598,A -85,B 0,C 180,E1 -5609.752,E2 -5609.752} C_VEL
LIN {X 0,Y 509.87,Z 281.596,A -85,B 0,C 180,E1 -5612.775,E2 -5612.775} C_VEL
LIN {X 0,Y 509.816,Z 281.605,A -85,B 0,C 180,E1 -5615.579,E2 -5615.579} C_VEL
LIN {X 0,Y 509.845,Z 281.605,A -85,B 0,C 180,E1 -5618.339,E2 -5618.339} C_VEL
LIN {X 0,Y 509.851,Z 281.605,A -85,B 0,C 180,E1 -5621.426,E2 -5621.426} C_VEL
LIN {X 0,Y 509.852,Z 281.602,A -85,B 0,C 180,E1 -5624.669,E2 -5624.669} C_VEL
LIN {X 0,Y 509.821,Z 281.79,A -85,B 0,C 180,E1 -5627.51,E2 -5627.51} C_VEL
LIN {X 0,Y 510.013,Z 284.793,A -85,B 0,C 180,E1 -5629.636,E2 -5629.636} C_VEL
LIN {X 0,Y 509.93,Z 289.873,A -85,B 0,C 180,E1 -5633.07,E2 -5633.07} C_VEL
LIN {X 0,Y 509.89,Z 290.698,A -85,B 0,C 180,E1 -5633.614,E2 -5633.614} C_VEL
LIN {X 0,Y 509.211,Z 291.771,A -85,B 0,C 180,E1 -5634.262,E2 -5634.262} C_VEL
LIN {X 0,Y 506.332,Z 293.742,A -85,B 0,C 180,E1 -5635.309,E2 -5635.309} C_VEL
LIN {X 0,Y 503.881,Z 295.346,A -85,B 0,C 180,E1 -5636.152,E2 -5636.152} C_VEL
LIN {X 0,Y 502.802,Z 296.488,A -85,B 0,C 180,E1 -5636.806,E2 -5636.806} C_VEL
LIN {X 0,Y 502.7,Z 296.844,A -85,B 0,C 180,E1 -5637.027,E2 -5637.027} C_VEL
LIN {X 0,Y 502.584,Z 301.725,A -85,B 0,C 180,E1 -5640.111,E2 -5640.111} C_VEL
LIN {X 0,Y 502.483,Z 305.627,A -85,B 0,C 180,E1 -5642.513,E2 -5642.513} C_VEL
LIN {X 0,Y 502.401,Z 310.459,A -85,B 0,C 180,E1 -5645.405,E2 -5645.405} C_VEL
LIN {X 0,Y 502.289,Z 314.564,A -85,B 0,C 180,E1 -5647.804,E2 -5647.804} C_VEL
LIN {X 0,Y 502.279,Z 318.165,A -85,B 0,C 180,E1 -5649.866,E2 -5649.866} C_VEL
LIN {X 0,Y 506.474,Z 334.07,A -85,B 0,C 180,E1 -5650.361,E2 -5650.361} C_VEL
LIN {X 0,Y 507.243,Z 337.721,A -85,B 0,C 180,E1 -5650.496,E2 -5650.496} C_VEL
LIN {X 0,Y 506.85,Z 352.87,A -85,B 0,C 180,E1 -5651,E2 -5651} C_VEL
LIN {X 0,Y 506.233,Z 368.281,A -85,B 0,C 180,E1 -5651.694,E2 -5651.694} C_VEL
LIN {X 0,Y 505.646,Z 382.31,A -85,B 0,C 180,E1 -5652.509,E2 -5652.509} C_VEL
LIN {X 0,Y 505.084,Z 395.131,A -85,B 0,C 180,E1 -5653.427,E2 -5653.427} C_VEL
LIN {X 0,Y 504.455,Z 407.386,A -85,B 0,C 180,E1 -5654.484,E2 -5654.484} C_VEL
LIN {X 0,Y 503.91,Z 418.839,A -85,B 0,C 180,E1 -5655.668,E2 -5655.668} C_VEL
LIN {X 0,Y 503.421,Z 428.82,A -85,B 0,C 180,E1 -5656.888,E2 -5656.888} C_VEL
LIN {X 0,Y 502.985,Z 437.505,A -85,B 0,C 180,E1 -5658.139,E2 -5658.139} C_VEL
LIN {X 0,Y 502.741,Z 445.596,A -85,B 0,C 180,E1 -5659.53,E2 -5659.53} C_VEL
LIN {X 0,Y 502.444,Z 453.398,A -85,B 0,C 180,E1 -5661.15,E2 -5661.15} C_VEL
LIN {X 0,Y 502.245,Z 459.613,A -85,B 0,C 180,E1 -5662.765,E2 -5662.765} C_VEL
LIN {X 0,Y 502.215,Z 464.414,A -85,B 0,C 180,E1 -5664.379,E2 -5664.379} C_VEL
LIN {X 0,Y 502.099,Z 467.936,A -85,B 0,C 180,E1 -5665.987,E2 -5665.987} C_VEL
LIN {X 0,Y 502.088,Z 470.267,A -85,B 0,C 180,E1 -5667.594,E2 -5667.594} C_VEL
LIN {X 0,Y 501.987,Z 471.462,A -85,B 0,C 180,E1 -5669.198,E2 -5669.198} C_VEL
LIN {X 0,Y 501.988,Z 471.48,A -85,B 0,C 180,E1 -5670.802,E2 -5670.802} C_VEL
LIN {X 0,Y 502.089,Z 470.36,A -85,B 0,C 180,E1 -5672.407,E2 -5672.407} C_VEL
LIN {X 0,Y 502.099,Z 468.101,A -85,B 0,C 180,E1 -5674.013,E2 -5674.013} C_VEL
LIN {X 0,Y 502.207,Z 464.649,A -85,B 0,C 180,E1 -5675.622,E2 -5675.622} C_VEL
LIN {X 0,Y 502.245,Z 459.923,A -85,B 0,C 180,E1 -5677.235,E2 -5677.235} C_VEL
LIN {X 0,Y 502.44,Z 453.799,A -85,B 0,C 180,E1 -5678.851,E2 -5678.851} C_VEL
LIN {X 0,Y 502.738,Z 446.09,A -85,B 0,C 180,E1 -5680.471,E2 -5680.471} C_VEL
LIN {X 0,Y 502.98,Z 438.092,A -85,B 0,C 180,E1 -5681.858,E2 -5681.858} C_VEL
LIN {X 0,Y 503.443,Z 427.976,A -85,B 0,C 180,E1 -5683.317,E2 -5683.317} C_VEL
LIN {X 0,Y 503.949,Z 417.83,A -85,B 0,C 180,E1 -5684.538,E2 -5684.538} C_VEL
LIN {X 0,Y 504.503,Z 406.818,A -85,B 0,C 180,E1 -5685.659,E2 -5685.659} C_VEL
LIN {X 0,Y 505.087,Z 394.942,A -85,B 0,C 180,E1 -5686.678,E2 -5686.678} C_VEL
LIN {X 0,Y 505.681,Z 382.088,A -85,B 0,C 180,E1 -5687.595,E2 -5687.595} C_VEL
LIN {X 0,Y 506.268,Z 367.994,A -85,B 0,C 180,E1 -5688.41,E2 -5688.41} C_VEL
LIN {X 0,Y 506.804,Z 353.107,A -85,B 0,C 180,E1 -5689.082,E2 -5689.082} C_VEL
LIN {X 0,Y 507.248,Z 338.037,A -85,B 0,C 180,E1 -5689.584,E2 -5689.584} C_VEL
LIN {X 0,Y 504.431,Z 326.097,A -85,B 0,C 180,E1 -5689.996,E2 -5689.996} C_VEL
LIN {X 0,Y 502.284,Z 318.147,A -85,B 0,C 180,E1 -5690.225,E2 -5690.225} C_VEL
LIN {X 0,Y 502.336,Z 313.265,A -85,B 0,C 180,E1 -5693.063,E2 -5693.063} C_VEL
LIN {X 0,Y 502.415,Z 308.816,A -85,B 0,C 180,E1 -5695.699,E2 -5695.699} C_VEL
LIN {X 0,Y 502.514,Z 304.36,A -85,B 0,C 180,E1 -5698.393,E2 -5698.393} C_VEL
LIN {X 0,Y 502.634,Z 299.392,A -85,B 0,C 180,E1 -5701.469,E2 -5701.469} C_VEL
LIN {X 0,Y 502.791,Z 294.721,A -85,B 0,C 180,E1 -5704.442,E2 -5704.442} C_VEL
LIN {X 0,Y 502.898,Z 290.54,A -85,B 0,C 180,E1 -5707.196,E2 -5707.196} C_VEL
LIN {X 0,Y 502.979,Z 286.453,A -85,B 0,C 180,E1 -5709.997,E2 -5709.997} C_VEL
LIN {X 0,Y 502.858,Z 283.347,A -85,B 0,C 180,E1 -5712.206,E2 -5712.206} C_VEL
LIN {X 0,Y 502.755,Z 282.487,A -85,B 0,C 180,E1 -5713.372,E2 -5713.372} C_VEL
LIN {X 0,Y 502.789,Z 282.485,A -85,B 0,C 180,E1 -5715.661,E2 -5715.661} C_VEL
LIN {X 0,Y 502.817,Z 282.478,A -85,B 0,C 180,E1 -5719.005,E2 -5719.005} C_VEL
LIN {X 0,Y 502.792,Z 282.483,A -85,B 0,C 180,E1 -5722.046,E2 -5722.046} C_VEL
LIN {X 0,Y 502.794,Z 282.484,A -85,B 0,C 180,E1 -5725.034,E2 -5725.034} C_VEL
LIN {X 0,Y 502.781,Z 282.485,A -85,B 0,C 180,E1 -5727.915,E2 -5727.915} C_VEL
LIN {X 0,Y 502.81,Z 282.479,A -85,B 0,C 180,E1 -5730.711,E2 -5730.711} C_VEL
LIN {X 0,Y 502.841,Z 282.472,A -85,B 0,C 180,E1 -5733.443,E2 -5733.443} C_VEL
LIN {X 0,Y 502.777,Z 282.482,A -85,B 0,C 180,E1 -5736.085,E2 -5736.085} C_VEL
LIN {X 0,Y 502.777,Z 282.485,A -85,B 0,C 180,E1 -5738.688,E2 -5738.688} C_VEL
LIN {X 0,Y 502.826,Z 282.474,A -85,B 0,C 180,E1 -5741.248,E2 -5741.248} C_VEL
LIN {X 0,Y 502.818,Z 282.475,A -85,B 0,C 180,E1 -5743.767,E2 -5743.767} C_VEL
LIN {X 0,Y 502.818,Z 282.48,A -85,B 0,C 180,E1 -5746.254,E2 -5746.254} C_VEL
LIN {X 0,Y 502.874,Z 282.469,A -85,B 0,C 180,E1 -5748.717,E2 -5748.717} C_VEL
LIN {X 0,Y 502.877,Z 282.469,A -85,B 0,C 180,E1 -5751.966,E2 -5751.966} C_VEL
LIN {X 0,Y 502.922,Z 282.464,A -85,B 0,C 180,E1 -5754.386,E2 -5754.386} C_VEL
LIN {X 0,Y 503.023,Z 282.45,A -85,B 0,C 180,E1 -5757.598,E2 -5757.598} C_VEL
LIN {X 0,Y 502.985,Z 282.455,A -85,B 0,C 180,E1 -5760.801,E2 -5760.801} C_VEL
LIN {X 0,Y 502.897,Z 282.47,A -85,B 0,C 180,E1 -5763.204,E2 -5763.204} C_VEL
LIN {X 0,Y 502.877,Z 282.47,A -85,B 0,C 180,E1 -5766.419,E2 -5766.419} C_VEL
LIN {X 0,Y 502.869,Z 282.471,A -85,B 0,C 180,E1 -5768.843,E2 -5768.843} C_VEL
LIN {X 0,Y 502.842,Z 282.476,A -85,B 0,C 180,E1 -5772.102,E2 -5772.102} C_VEL
LIN {X 0,Y 502.845,Z 282.477,A -85,B 0,C 180,E1 -5775.4,E2 -5775.4} C_VEL
LIN {X 0,Y 502.842,Z 282.475,A -85,B 0,C 180,E1 -5778.122,E2 -5778.122} C_VEL
LIN {X 0,Y 502.825,Z 282.475,A -85,B 0,C 180,E1 -5780.536,E2 -5780.536} C_VEL
LIN {X 0,Y 502.787,Z 282.484,A -85,B 0,C 180,E1 -5783.041,E2 -5783.041} C_VEL
LIN {X 0,Y 502.836,Z 282.475,A -85,B 0,C 180,E1 -5785.676,E2 -5785.676} C_VEL
LIN {X 0,Y 502.833,Z 282.475,A -85,B 0,C 180,E1 -5788.373,E2 -5788.373} C_VEL
LIN {X 0,Y 502.789,Z 282.482,A -85,B 0,C 180,E1 -5791.499,E2 -5791.499} C_VEL
LIN {X 0,Y 502.799,Z 282.484,A -85,B 0,C 180,E1 -5793.994,E2 -5793.994} C_VEL
LIN {X 0,Y 502.774,Z 282.486,A -85,B 0,C 180,E1 -5797.178,E2 -5797.178} C_VEL
LIN {X 0,Y 502.785,Z 282.484,A -85,B 0,C 180,E1 -5800.015,E2 -5800.015} C_VEL
LIN {X 0,Y 502.8,Z 282.48,A -85,B 0,C 180,E1 -5802.199,E2 -5802.199} C_VEL
LIN {X 0,Y 502.801,Z 282.486,A -85,B 0,C 180,E1 -5805.468,E2 -5805.468} C_VEL
LIN {X 0,Y 502.845,Z 282.537,A -85,B 0,C 180,E1 -5806.172,E2 -5806.172} C_VEL
LIN {X 0,Y 503.326,Z 286.949,A -85,B 0,C 180,E1 -5808.939,E2 -5808.939} C_VEL
LIN {X 0,Y 503.151,Z 292.319,A -85,B 0,C 180,E1 -5812.078,E2 -5812.078} C_VEL
LIN {X 0,Y 503.008,Z 297.635,A -85,B 0,C 180,E1 -5815.051,E2 -5815.051} C_VEL
LIN {X 0,Y 502.806,Z 302.943,A -85,B 0,C 180,E1 -5817.917,E2 -5817.917} C_VEL
LIN {X 0,Y 502.668,Z 308.261,A -85,B 0,C 180,E1 -5820.702,E2 -5820.702} C_VEL
LIN {X 0,Y 502.532,Z 313.795,A -85,B 0,C 180,E1 -5823.515,E2 -5823.515} C_VEL
LIN {X 0,Y 502.42,Z 318.938,A -85,B 0,C 180,E1 -5826.068,E2 -5826.068} C_VEL
LIN {X 0,Y 502.329,Z 324.29,A -85,B 0,C 180,E1 -5828.669,E2 -5828.669} C_VEL
LIN {X 0,Y 502.359,Z 326.638,A -85,B 0,C 180,E1 -5829.798,E2 -5829.798} C_VEL
LIN {X 0,Y 506.904,Z 345.086,A -85,B 0,C 180,E1 -5830.383,E2 -5830.383} C_VEL
LIN {X 0,Y 507.201,Z 347.753,A -85,B 0,C 180,E1 -5830.471,E2 -5830.471} C_VEL
LIN {X 0,Y 506.82,Z 360.928,A -85,B 0,C 180,E1 -5830.904,E2 -5830.904} C_VEL
LIN {X 0,Y 506.303,Z 374.492,A -85,B 0,C 180,E1 -5831.486,E2 -5831.486} C_VEL
LIN {X 0,Y 505.689,Z 389.197,A -85,B 0,C 180,E1 -5832.301,E2 -5832.301} C_VEL
LIN {X 0,Y 505.099,Z 402.501,A -85,B 0,C 180,E1 -5833.219,E2 -5833.219} C_VEL
LIN {X 0,Y 504.488,Z 415.741,A -85,B 0,C 180,E1 -5834.335,E2 -5834.335} C_VEL
LIN {X 0,Y 503.91,Z 426.928,A -85,B 0,C 180,E1 -5835.461,E2 -5835.461} C_VEL
LIN {X 0,Y 503.437,Z 437.158,A -85,B 0,C 180,E1 -5836.683,E2 -5836.683} C_VEL
LIN {X 0,Y 502.935,Z 447.54,A -85,B 0,C 180,E1 -5838.165,E2 -5838.165} C_VEL
LIN {X 0,Y 502.716,Z 455.458,A -85,B 0,C 180,E1 -5839.529,E2 -5839.529} C_VEL
LIN {X 0,Y 502.417,Z 463.253,A -85,B 0,C 180,E1 -5841.148,E2 -5841.148} C_VEL
LIN {X 0,Y 502.244,Z 469.454,A -85,B 0,C 180,E1 -5842.765,E2 -5842.765} C_VEL
LIN {X 0,Y 502.195,Z 474.249,A -85,B 0,C 180,E1 -5844.378,E2 -5844.378} C_VEL
LIN {X 0,Y 502.094,Z 477.76,A -85,B 0,C 180,E1 -5845.987,E2 -5845.987} C_VEL
LIN {X 0,Y 502.062,Z 480.07,A -85,B 0,C 180,E1 -5847.593,E2 -5847.593} C_VEL
LIN {X 0,Y 501.987,Z 481.232,A -85,B 0,C 180,E1 -5849.198,E2 -5849.198} C_VEL
LIN {X 0,Y 501.987,Z 481.231,A -85,B 0,C 180,E1 -5850.802,E2 -5850.802} C_VEL
LIN {X 0,Y 502.062,Z 480.066,A -85,B 0,C 180,E1 -5852.406,E2 -5852.406} C_VEL
LIN {X 0,Y 502.094,Z 477.756,A -85,B 0,C 180,E1 -5854.013,E2 -5854.013} C_VEL
LIN {X 0,Y 502.196,Z 474.251,A -85,B 0,C 180,E1 -5855.621,E2 -5855.621} C_VEL
LIN {X 0,Y 502.245,Z 469.46,A -85,B 0,C 180,E1 -5857.235,E2 -5857.235} C_VEL
LIN {X 0,Y 502.416,Z 463.252,A -85,B 0,C 180,E1 -5858.851,E2 -5858.851} C_VEL
LIN {X 0,Y 502.715,Z 455.455,A -85,B 0,C 180,E1 -5860.471,E2 -5860.471} C_VEL
LIN {X 0,Y 502.967,Z 447.425,A -85,B 0,C 180,E1 -5861.852,E2 -5861.852} C_VEL
LIN {X 0,Y 503.436,Z 437.163,A -85,B 0,C 180,E1 -5863.317,E2 -5863.317} C_VEL
LIN {X 0,Y 503.909,Z 426.935,A -85,B 0,C 180,E1 -5864.539,E2 -5864.539} C_VEL
LIN {X 0,Y 504.536,Z 414.407,A -85,B 0,C 180,E1 -5865.793,E2 -5865.793} C_VEL
LIN {X 0,Y 505.175,Z 401.183,A -85,B 0,C 180,E1 -5866.882,E2 -5866.882} C_VEL
LIN {X 0,Y 505.779,Z 387.577,A -85,B 0,C 180,E1 -5867.8,E2 -5867.8} C_VEL
LIN {X 0,Y 506.409,Z 373.485,A -85,B 0,C 180,E1 -5868.561,E2 -5868.561} C_VEL
LIN {X 0,Y 506.89,Z 358.822,A -85,B 0,C 180,E1 -5869.179,E2 -5869.179} C_VEL
LIN {X 0,Y 507.111,Z 345.819,A -85,B 0,C 180,E1 -5869.588,E2 -5869.588} C_VEL
LIN {X 0,Y 503.208,Z 330.403,A -85,B 0,C 180,E1 -5870.088,E2 -5870.088} C_VEL
LIN {X 0,Y 502.364,Z 326.671,A -85,B 0,C 180,E1 -5870.194,E2 -5870.194} C_VEL
LIN {X 0,Y 502.384,Z 320.76,A -85,B 0,C 180,E1 -5873.06,E2 -5873.06} C_VEL
LIN {X 0,Y 502.473,Z 315.443,A -85,B 0,C 180,E1 -5875.695,E2 -5875.695} C_VEL
LIN {X 0,Y 502.627,Z 310.101,A -85,B 0,C 180,E1 -5878.385,E2 -5878.385} C_VEL
LIN {X 0,Y 502.779,Z 304.749,A -85,B 0,C 180,E1 -5881.144,E2 -5881.144} C_VEL
LIN {X 0,Y 502.938,Z 299.411,A -85,B 0,C 180,E1 -5883.983,E2 -5883.983} C_VEL
LIN {X 0,Y 503.091,Z 294.089,A -85,B 0,C 180,E1 -5886.919,E2 -5886.919} C_VEL
LIN {X 0,Y 503.265,Z 288.779,A -85,B 0,C 180,E1 -5889.968,E2 -5889.968} C_VEL
LIN {X 0,Y 503.172,Z 285.25,A -85,B 0,C 180,E1 -5892.099,E2 -5892.099} C_VEL
LIN {X 0,Y 502.844,Z 282.472,A -85,B 0,C 180,E1 -5893.954,E2 -5893.954} C_VEL
LIN {X 0,Y 502.766,Z 282.486,A -85,B 0,C 180,E1 -5896.768,E2 -5896.768} C_VEL
LIN {X 0,Y 502.812,Z 282.48,A -85,B 0,C 180,E1 -5899.004,E2 -5899.004} C_VEL
LIN {X 0,Y 502.787,Z 282.483,A -85,B 0,C 180,E1 -5902.046,E2 -5902.046} C_VEL
LIN {X 0,Y 502.789,Z 282.484,A -85,B 0,C 180,E1 -5905.033,E2 -5905.033} C_VEL
LIN {X 0,Y 502.78,Z 282.487,A -85,B 0,C 180,E1 -5907.915,E2 -5907.915} C_VEL
LIN {X 0,Y 502.814,Z 282.481,A -85,B 0,C 180,E1 -5910.712,E2 -5910.712} C_VEL
LIN {X 0,Y 502.854,Z 282.473,A -85,B 0,C 180,E1 -5913.439,E2 -5913.439} C_VEL
LIN {X 0,Y 502.783,Z 282.48,A -85,B 0,C 180,E1 -5916.086,E2 -5916.086} C_VEL
LIN {X 0,Y 502.775,Z 282.485,A -85,B 0,C 180,E1 -5918.689,E2 -5918.689} C_VEL
LIN {X 0,Y 502.822,Z 282.476,A -85,B 0,C 180,E1 -5921.248,E2 -5921.248} C_VEL
LIN {X 0,Y 502.813,Z 282.477,A -85,B 0,C 180,E1 -5923.767,E2 -5923.767} C_VEL
LIN {X 0,Y 502.818,Z 282.481,A -85,B 0,C 180,E1 -5926.254,E2 -5926.254} C_VEL
LIN {X 0,Y 502.874,Z 282.468,A -85,B 0,C 180,E1 -5928.717,E2 -5928.717} C_VEL
LIN {X 0,Y 502.872,Z 282.47,A -85,B 0,C 180,E1 -5931.966,E2 -5931.966} C_VEL
LIN {X 0,Y 502.919,Z 282.462,A -85,B 0,C 180,E1 -5934.386,E2 -5934.386} C_VEL
LIN {X 0,Y 503.019,Z 282.449,A -85,B 0,C 180,E1 -5937.598,E2 -5937.598} C_VEL
LIN {X 0,Y 503.001,Z 282.453,A -85,B 0,C 180,E1 -5940.801,E2 -5940.801} C_VEL
LIN {X 0,Y 502.895,Z 282.469,A -85,B 0,C 180,E1 -5943.205,E2 -5943.205} C_VEL
LIN {X 0,Y 502.873,Z 282.471,A -85,B 0,C 180,E1 -5946.42,E2 -5946.42} C_VEL
LIN {X 0,Y 502.865,Z 282.47,A -85,B 0,C 180,E1 -5948.844,E2 -5948.844} C_VEL
LIN {X 0,Y 502.837,Z 282.475,A -85,B 0,C 180,E1 -5952.102,E2 -5952.102} C_VEL
LIN {X 0,Y 502.84,Z 282.477,A -85,B 0,C 180,E1 -5955.4,E2 -5955.4} C_VEL
LIN {X 0,Y 502.838,Z 282.475,A -85,B 0,C 180,E1 -5958.123,E2 -5958.123} C_VEL
LIN {X 0,Y 502.821,Z 282.475,A -85,B 0,C 180,E1 -5960.537,E2 -5960.537} C_VEL
LIN {X 0,Y 502.786,Z 282.484,A -85,B 0,C 180,E1 -5963.041,E2 -5963.041} C_VEL
LIN {X 0,Y 502.832,Z 282.475,A -85,B 0,C 180,E1 -5965.676,E2 -5965.676} C_VEL
LIN {X 0,Y 502.829,Z 282.473,A -85,B 0,C 180,E1 -5968.373,E2 -5968.373} C_VEL
LIN {X 0,Y 502.79,Z 282.478,A -85,B 0,C 180,E1 -5971.5,E2 -5971.5} C_VEL
LIN {X 0,Y 502.796,Z 282.479,A -85,B 0,C 180,E1 -5973.995,E2 -5973.995} C_VEL
LIN {X 0,Y 502.771,Z 282.482,A -85,B 0,C 180,E1 -5977.178,E2 -5977.178} C_VEL
LIN {X 0,Y 502.783,Z 282.484,A -85,B 0,C 180,E1 -5980.016,E2 -5980.016} C_VEL
LIN {X 0,Y 502.798,Z 282.48,A -85,B 0,C 180,E1 -5982.2,E2 -5982.2} C_VEL
LIN {X 0,Y 502.796,Z 282.48,A -85,B 0,C 180,E1 -5985.469,E2 -5985.469} C_VEL
LIN {X 0,Y 502.751,Z 282.488,A -85,B 0,C 180,E1 -5986.768,E2 -5986.768} C_VEL
LIN {X 0,Y 502.859,Z 283.317,A -85,B 0,C 180,E1 -5987.868,E2 -5987.868} C_VEL
LIN {X 0,Y 502.972,Z 286.632,A -85,B 0,C 180,E1 -5990.221,E2 -5990.221} C_VEL
LIN {X 0,Y 502.888,Z 290.788,A -85,B 0,C 180,E1 -5993.064,E2 -5993.064} C_VEL
LIN {X 0,Y 502.762,Z 295.254,A -85,B 0,C 180,E1 -5996.004,E2 -5996.004} C_VEL
LIN {X 0,Y 502.7,Z 296.844,A -85,B 0,C 180,E1 -5997.027,E2 -5997.027} C_VEL
LIN {X 0,Y 501.994,Z 297.951,A -85,B 0,C 180,E1 -5997.684,E2 -5997.684} C_VEL
LIN {X 0,Y 499.115,Z 299.953,A -85,B 0,C 180,E1 -5998.745,E2 -5998.745} C_VEL
LIN {X 0,Y 496.681,Z 301.577,A -85,B 0,C 180,E1 -5999.599,E2 -5999.599} C_VEL
LIN {X 0,Y 495.605,Z 302.744,A -85,B 0,C 180,E1 -6000.261,E2 -6000.261} C_VEL
LIN {X 0,Y 495.501,Z 303.111,A -85,B 0,C 180,E1 -6000.486,E2 -6000.486} C_VEL
LIN {X 0,Y 495.401,Z 307.724,A -85,B 0,C 180,E1 -6003.348,E2 -6003.348} C_VEL
LIN {X 0,Y 495.309,Z 311.639,A -85,B 0,C 180,E1 -6005.703,E2 -6005.703} C_VEL
LIN {X 0,Y 495.191,Z 316.114,A -85,B 0,C 180,E1 -6008.346,E2 -6008.346} C_VEL
LIN {X 0,Y 495.192,Z 318.181,A -85,B 0,C 180,E1 -6009.555,E2 -6009.555} C_VEL
LIN {X 0,Y 499.774,Z 335.428,A -85,B 0,C 180,E1 -6010.123,E2 -6010.123} C_VEL
LIN {X 0,Y 500.526,Z 339.374,A -85,B 0,C 180,E1 -6010.269,E2 -6010.269} C_VEL
LIN {X 0,Y 500.097,Z 354.544,A -85,B 0,C 180,E1 -6010.799,E2 -6010.799} C_VEL
LIN {X 0,Y 499.48,Z 368.363,A -85,B 0,C 180,E1 -6011.438,E2 -6011.438} C_VEL
LIN {X 0,Y 498.86,Z 382.39,A -85,B 0,C 180,E1 -6012.263,E2 -6012.263} C_VEL
LIN {X 0,Y 498.243,Z 395.209,A -85,B 0,C 180,E1 -6013.193,E2 -6013.193} C_VEL
LIN {X 0,Y 497.573,Z 407.62,A -85,B 0,C 180,E1 -6014.279,E2 -6014.279} C_VEL
LIN {X 0,Y 496.974,Z 418.914,A -85,B 0,C 180,E1 -6015.463,E2 -6015.463} C_VEL
LIN {X 0,Y 496.462,Z 428.894,A -85,B 0,C 180,E1 -6016.701,E2 -6016.701} C_VEL
LIN {X 0,Y 495.972,Z 438.066,A -85,B 0,C 180,E1 -6018.047,E2 -6018.047} C_VEL
LIN {X 0,Y 495.736,Z 445.669,A -85,B 0,C 180,E1 -6019.38,E2 -6019.38} C_VEL
LIN {X 0,Y 495.388,Z 453.471,A -85,B 0,C 180,E1 -6021.022,E2 -6021.022} C_VEL
LIN {X 0,Y 495.171,Z 459.684,A -85,B 0,C 180,E1 -6022.662,E2 -6022.662} C_VEL
LIN {X 0,Y 495.127,Z 464.485,A -85,B 0,C 180,E1 -6024.298,E2 -6024.298} C_VEL
LIN {X 0,Y 494.998,Z 468.006,A -85,B 0,C 180,E1 -6025.93,E2 -6025.93} C_VEL
LIN {X 0,Y 494.995,Z 470.337,A -85,B 0,C 180,E1 -6027.559,E2 -6027.559} C_VEL
LIN {X 0,Y 494.907,Z 471.531,A -85,B 0,C 180,E1 -6029.187,E2 -6029.187} C_VEL
LIN {X 0,Y 494.908,Z 471.549,A -85,B 0,C 180,E1 -6030.814,E2 -6030.814} C_VEL
LIN {X 0,Y 494.995,Z 470.428,A -85,B 0,C 180,E1 -6032.441,E2 -6032.441} C_VEL
LIN {X 0,Y 494.998,Z 468.169,A -85,B 0,C 180,E1 -6034.071,E2 -6034.071} C_VEL
LIN {X 0,Y 495.116,Z 464.716,A -85,B 0,C 180,E1 -6035.703,E2 -6035.703} C_VEL
LIN {X 0,Y 495.171,Z 459.99,A -85,B 0,C 180,E1 -6037.339,E2 -6037.339} C_VEL
LIN {X 0,Y 495.383,Z 453.866,A -85,B 0,C 180,E1 -6038.978,E2 -6038.978} C_VEL
LIN {X 0,Y 495.731,Z 446.156,A -85,B 0,C 180,E1 -6040.621,E2 -6040.621} C_VEL
LIN {X 0,Y 496.031,Z 437.428,A -85,B 0,C 180,E1 -6042.143,E2 -6042.143} C_VEL
LIN {X 0,Y 496.498,Z 428.041,A -85,B 0,C 180,E1 -6043.507,E2 -6043.507} C_VEL
LIN {X 0,Y 497.037,Z 417.894,A -85,B 0,C 180,E1 -6044.745,E2 -6044.745} C_VEL
LIN {X 0,Y 497.663,Z 406.102,A -85,B 0,C 180,E1 -6045.957,E2 -6045.957} C_VEL
LIN {X 0,Y 498.311,Z 393.715,A -85,B 0,C 180,E1 -6047.017,E2 -6047.017} C_VEL
LIN {X 0,Y 498.966,Z 380.568,A -85,B 0,C 180,E1 -6047.946,E2 -6047.946} C_VEL
LIN {X 0,Y 499.541,Z 368.05,A -85,B 0,C 180,E1 -6048.667,E2 -6048.667} C_VEL
LIN {X 0,Y 500.072,Z 353.964,A -85,B 0,C 180,E1 -6049.316,E2 -6049.316} C_VEL
LIN {X 0,Y 500.456,Z 338.27,A -85,B 0,C 180,E1 -6049.855,E2 -6049.855} C_VEL
LIN {X 0,Y 496.504,Z 323.116,A -85,B 0,C 180,E1 -6050.383,E2 -6050.383} C_VEL
LIN {X 0,Y 495.198,Z 318.167,A -85,B 0,C 180,E1 -6050.552,E2 -6050.552} C_VEL
LIN {X 0,Y 495.269,Z 313.327,A -85,B 0,C 180,E1 -6053.411,E2 -6053.411} C_VEL
LIN {X 0,Y 495.36,Z 308.871,A -85,B 0,C 180,E1 -6056.092,E2 -6056.092} C_VEL
LIN {X 0,Y 495.455,Z 304.411,A -85,B 0,C 180,E1 -6058.835,E2 -6058.835} C_VEL
LIN {X 0,Y 495.593,Z 299.867,A -85,B 0,C 180,E1 -6061.695,E2 -6061.695} C_VEL
LIN {X 0,Y 495.767,Z 295.227,A -85,B 0,C 180,E1 -6064.693,E2 -6064.693} C_VEL
LIN {X 0,Y 495.845,Z 290.965,A -85,B 0,C 180,E1 -6067.551,E2 -6067.551} C_VEL
LIN {X 0,Y 495.961,Z 286.477,A -85,B 0,C 180,E1 -6070.68,E2 -6070.68} C_VEL
LIN {X 0,Y 495.728,Z 283.48,A -85,B 0,C 180,E1 -6072.882,E2 -6072.882} C_VEL
LIN {X 0,Y 495.733,Z 283.363,A -85,B 0,C 180,E1 -6075.999,E2 -6075.999} C_VEL
LIN {X 0,Y 495.765,Z 283.355,A -85,B 0,C 180,E1 -6079.3,E2 -6079.3} C_VEL
LIN {X 0,Y 495.727,Z 283.361,A -85,B 0,C 180,E1 -6082.438,E2 -6082.438} C_VEL
LIN {X 0,Y 495.774,Z 283.355,A -85,B 0,C 180,E1 -6085.456,E2 -6085.456} C_VEL
LIN {X 0,Y 495.753,Z 283.358,A -85,B 0,C 180,E1 -6088.363,E2 -6088.363} C_VEL
LIN {X 0,Y 495.752,Z 283.357,A -85,B 0,C 180,E1 -6091.514,E2 -6091.514} C_VEL
LIN {X 0,Y 495.756,Z 283.358,A -85,B 0,C 180,E1 -6093.93,E2 -6093.93} C_VEL
LIN {X 0,Y 495.758,Z 283.359,A -85,B 0,C 180,E1 -6097.139,E2 -6097.139} C_VEL
LIN {X 0,Y 495.767,Z 283.358,A -85,B 0,C 180,E1 -6100.109,E2 -6100.109} C_VEL
LIN {X 0,Y 495.783,Z 283.353,A -85,B 0,C 180,E1 -6102.681,E2 -6102.681} C_VEL
LIN {X 0,Y 495.782,Z 283.353,A -85,B 0,C 180,E1 -6105.217,E2 -6105.217} C_VEL
LIN {X 0,Y 495.848,Z 283.344,A -85,B 0,C 180,E1 -6108.555,E2 -6108.555} C_VEL
LIN {X 0,Y 495.834,Z 283.346,A -85,B 0,C 180,E1 -6111.851,E2 -6111.851} C_VEL
LIN {X 0,Y 495.837,Z 283.347,A -85,B 0,C 180,E1 -6115.121,E2 -6115.121} C_VEL
LIN {X 0,Y 495.991,Z 283.326,A -85,B 0,C 180,E1 -6117.564,E2 -6117.564} C_VEL
LIN {X 0,Y 495.937,Z 283.333,A -85,B 0,C 180,E1 -6120.812,E2 -6120.812} C_VEL
LIN {X 0,Y 495.991,Z 283.326,A -85,B 0,C 180,E1 -6122.436,E2 -6122.436} C_VEL
LIN {X 0,Y 495.877,Z 283.341,A -85,B 0,C 180,E1 -6125.694,E2 -6125.694} C_VEL
LIN {X 0,Y 495.838,Z 283.348,A -85,B 0,C 180,E1 -6128.97,E2 -6128.97} C_VEL
LIN {X 0,Y 495.824,Z 283.35,A -85,B 0,C 180,E1 -6132.035,E2 -6132.035} C_VEL
LIN {X 0,Y 495.82,Z 283.351,A -85,B 0,C 180,E1 -6135.452,E2 -6135.452} C_VEL
LIN {X 0,Y 495.803,Z 283.353,A -85,B 0,C 180,E1 -6138.247,E2 -6138.247} C_VEL
LIN {X 0,Y 495.77,Z 283.354,A -85,B 0,C 180,E1 -6140.756,E2 -6140.756} C_VEL
LIN {X 0,Y 495.744,Z 283.358,A -85,B 0,C 180,E1 -6143.387,E2 -6143.387} C_VEL
LIN {X 0,Y 495.787,Z 283.356,A -85,B 0,C 180,E1 -6146.068,E2 -6146.068} C_VEL
LIN {X 0,Y 495.765,Z 283.358,A -85,B 0,C 180,E1 -6148.815,E2 -6148.815} C_VEL
LIN {X 0,Y 495.751,Z 283.36,A -85,B 0,C 180,E1 -6151.725,E2 -6151.725} C_VEL
LIN {X 0,Y 495.764,Z 283.359,A -85,B 0,C 180,E1 -6154.694,E2 -6154.694} C_VEL
LIN {X 0,Y 495.726,Z 283.363,A -85,B 0,C 180,E1 -6157.562,E2 -6157.562} C_VEL
LIN {X 0,Y 495.756,Z 283.359,A -85,B 0,C 180,E1 -6160.047,E2 -6160.047} C_VEL
LIN {X 0,Y 495.714,Z 283.366,A -85,B 0,C 180,E1 -6162.884,E2 -6162.884} C_VEL
LIN {X 0,Y 495.797,Z 283.478,A -85,B 0,C 180,E1 -6166.006,E2 -6166.006} C_VEL
LIN {X 0,Y 496.258,Z 287.59,A -85,B 0,C 180,E1 -6168.641,E2 -6168.641} C_VEL
LIN {X 0,Y 496.179,Z 292.288,A -85,B 0,C 180,E1 -6171.448,E2 -6171.448} C_VEL
LIN {X 0,Y 495.999,Z 297.597,A -85,B 0,C 180,E1 -6174.483,E2 -6174.483} C_VEL
LIN {X 0,Y 495.803,Z 302.898,A -85,B 0,C 180,E1 -6177.408,E2 -6177.408} C_VEL
LIN {X 0,Y 495.656,Z 308.217,A -85,B 0,C 180,E1 -6180.247,E2 -6180.247} C_VEL
LIN {X 0,Y 495.48,Z 314.174,A -85,B 0,C 180,E1 -6183.33,E2 -6183.33} C_VEL
LIN {X 0,Y 495.377,Z 318.876,A -85,B 0,C 180,E1 -6185.705,E2 -6185.705} C_VEL
LIN {X 0,Y 495.277,Z 324.22,A -85,B 0,C 180,E1 -6188.35,E2 -6188.35} C_VEL
LIN {X 0,Y 495.278,Z 326.581,A -85,B 0,C 180,E1 -6189.504,E2 -6189.504} C_VEL
LIN {X 0,Y 499.722,Z 344.238,A -85,B 0,C 180,E1 -6190.066,E2 -6190.066} C_VEL
LIN {X 0,Y 500.479,Z 348.448,A -85,B 0,C 180,E1 -6190.22,E2 -6190.22} C_VEL
LIN {X 0,Y 500.102,Z 362.714,A -85,B 0,C 180,E1 -6190.713,E2 -6190.713} C_VEL
LIN {X 0,Y 499.454,Z 376.412,A -85,B 0,C 180,E1 -6191.33,E2 -6191.33} C_VEL
LIN {X 0,Y 498.825,Z 390.711,A -85,B 0,C 180,E1 -6192.155,E2 -6192.155} C_VEL
LIN {X 0,Y 498.186,Z 403.724,A -85,B 0,C 180,E1 -6193.084,E2 -6193.084} C_VEL
LIN {X 0,Y 497.57,Z 416.048,A -85,B 0,C 180,E1 -6194.148,E2 -6194.148} C_VEL
LIN {X 0,Y 496.969,Z 426.858,A -85,B 0,C 180,E1 -6195.253,E2 -6195.253} C_VEL
LIN {X 0,Y 496.476,Z 437.088,A -85,B 0,C 180,E1 -6196.493,E2 -6196.493} C_VEL
LIN {X 0,Y 495.938,Z 446.899,A -85,B 0,C 180,E1 -6197.906,E2 -6197.906} C_VEL
LIN {X 0,Y 495.678,Z 455.388,A -85,B 0,C 180,E1 -6199.378,E2 -6199.378} C_VEL
LIN {X 0,Y 495.338,Z 463.183,A -85,B 0,C 180,E1 -6201.021,E2 -6201.021} C_VEL
LIN {X 0,Y 495.165,Z 469.384,A -85,B 0,C 180,E1 -6202.661,E2 -6202.661} C_VEL
LIN {X 0,Y 495.106,Z 474.179,A -85,B 0,C 180,E1 -6204.297,E2 -6204.297} C_VEL
LIN {X 0,Y 494.991,Z 477.691,A -85,B 0,C 180,E1 -6205.929,E2 -6205.929} C_VEL
LIN {X 0,Y 494.971,Z 480.001,A -85,B 0,C 180,E1 -6207.558,E2 -6207.558} C_VEL
LIN {X 0,Y 494.907,Z 481.163,A -85,B 0,C 180,E1 -6209.186,E2 -6209.186} C_VEL
LIN {X 0,Y 494.907,Z 481.163,A -85,B 0,C 180,E1 -6210.813,E2 -6210.813} C_VEL
LIN {X 0,Y 494.97,Z 479.997,A -85,B 0,C 180,E1 -6212.441,E2 -6212.441} C_VEL
LIN {X 0,Y 494.991,Z 477.687,A -85,B 0,C 180,E1 -6214.071,E2 -6214.071} C_VEL
LIN {X 0,Y 495.11,Z 474.182,A -85,B 0,C 180,E1 -6215.702,E2 -6215.702} C_VEL
LIN {X 0,Y 495.165,Z 469.39,A -85,B 0,C 180,E1 -6217.339,E2 -6217.339} C_VEL
LIN {X 0,Y 495.338,Z 463.183,A -85,B 0,C 180,E1 -6218.978,E2 -6218.978} C_VEL
LIN {X 0,Y 495.677,Z 455.385,A -85,B 0,C 180,E1 -6220.621,E2 -6220.621} C_VEL
LIN {X 0,Y 495.986,Z 446.723,A -85,B 0,C 180,E1 -6222.12,E2 -6222.12} C_VEL
LIN {X 0,Y 496.475,Z 437.093,A -85,B 0,C 180,E1 -6223.507,E2 -6223.507} C_VEL
LIN {X 0,Y 496.976,Z 426.865,A -85,B 0,C 180,E1 -6224.746,E2 -6224.746} C_VEL
LIN {X 0,Y 497.62,Z 414.909,A -85,B 0,C 180,E1 -6225.963,E2 -6225.963} C_VEL
LIN {X 0,Y 498.279,Z 402.445,A -85,B 0,C 180,E1 -6227.017,E2 -6227.017} C_VEL
LIN {X 0,Y 498.906,Z 389.131,A -85,B 0,C 180,E1 -6227.947,E2 -6227.947} C_VEL
LIN {X 0,Y 499.608,Z 374.435,A -85,B 0,C 180,E1 -6228.77,E2 -6228.77} C_VEL
LIN {X 0,Y 500.155,Z 359.225,A -85,B 0,C 180,E1 -6229.429,E2 -6229.429} C_VEL
LIN {X 0,Y 500.37,Z 347.103,A -85,B 0,C 180,E1 -6229.824,E2 -6229.824} C_VEL
LIN {X 0,Y 496.469,Z 331.444,A -85,B 0,C 180,E1 -6230.353,E2 -6230.353} C_VEL
LIN {X 0,Y 495.251,Z 326.563,A -85,B 0,C 180,E1 -6230.513,E2 -6230.513} C_VEL
LIN {X 0,Y 495.314,Z 320.699,A -85,B 0,C 180,E1 -6233.408,E2 -6233.408} C_VEL
LIN {X 0,Y 495.425,Z 315.39,A -85,B 0,C 180,E1 -6236.088,E2 -6236.088} C_VEL
LIN {X 0,Y 495.58,Z 310.051,A -85,B 0,C 180,E1 -6238.826,E2 -6238.826} C_VEL
LIN {X 0,Y 495.758,Z 304.536,A -85,B 0,C 180,E1 -6241.726,E2 -6241.726} C_VEL
LIN {X 0,Y 495.951,Z 299.015,A -85,B 0,C 180,E1 -6244.724,E2 -6244.724} C_VEL
LIN {X 0,Y 496.102,Z 294.049,A -85,B 0,C 180,E1 -6247.528,E2 -6247.528} C_VEL
LIN {X 0,Y 496.277,Z 288.751,A -85,B 0,C 180,E1 -6250.648,E2 -6250.648} C_VEL
LIN {X 0,Y 496.042,Z 285.211,A -85,B 0,C 180,E1 -6252.848,E2 -6252.848} C_VEL
LIN {X 0,Y 495.792,Z 283.351,A -85,B 0,C 180,E1 -6254.134,E2 -6254.134} C_VEL
LIN {X 0,Y 495.731,Z 283.363,A -85,B 0,C 180,E1 -6257.492,E2 -6257.492} C_VEL
LIN {X 0,Y 495.751,Z 283.361,A -85,B 0,C 180,E1 -6260.362,E2 -6260.362} C_VEL
LIN {X 0,Y 495.72,Z 283.365,A -85,B 0,C 180,E1 -6263.455,E2 -6263.455} C_VEL
LIN {X 0,Y 495.751,Z 283.363,A -85,B 0,C 180,E1 -6266.435,E2 -6266.435} C_VEL
LIN {X 0,Y 495.745,Z 283.364,A -85,B 0,C 180,E1 -6269.312,E2 -6269.312} C_VEL
LIN {X 0,Y 495.768,Z 283.357,A -85,B 0,C 180,E1 -6272.108,E2 -6272.108} C_VEL
LIN {X 0,Y 495.781,Z 283.353,A -85,B 0,C 180,E1 -6274.832,E2 -6274.832} C_VEL
LIN {X 0,Y 495.741,Z 283.358,A -85,B 0,C 180,E1 -6277.495,E2 -6277.495} C_VEL
LIN {X 0,Y 495.764,Z 283.358,A -85,B 0,C 180,E1 -6280.109,E2 -6280.109} C_VEL
LIN {X 0,Y 495.777,Z 283.353,A -85,B 0,C 180,E1 -6282.681,E2 -6282.681} C_VEL
LIN {X 0,Y 495.779,Z 283.352,A -85,B 0,C 180,E1 -6285.217,E2 -6285.217} C_VEL
LIN {X 0,Y 495.847,Z 283.343,A -85,B 0,C 180,E1 -6288.555,E2 -6288.555} C_VEL
LIN {X 0,Y 495.829,Z 283.346,A -85,B 0,C 180,E1 -6291.851,E2 -6291.851} C_VEL
LIN {X 0,Y 495.834,Z 283.346,A -85,B 0,C 180,E1 -6295.122,E2 -6295.122} C_VEL
LIN {X 0,Y 495.987,Z 283.325,A -85,B 0,C 180,E1 -6297.564,E2 -6297.564} C_VEL
LIN {X 0,Y 495.952,Z 283.331,A -85,B 0,C 180,E1 -6300.812,E2 -6300.812} C_VEL
LIN {X 0,Y 495.987,Z 283.326,A -85,B 0,C 180,E1 -6302.436,E2 -6302.436} C_VEL
LIN {X 0,Y 495.874,Z 283.342,A -85,B 0,C 180,E1 -6305.694,E2 -6305.694} C_VEL
LIN {X 0,Y 495.834,Z 283.347,A -85,B 0,C 180,E1 -6308.97,E2 -6308.97} C_VEL
LIN {X 0,Y 495.82,Z 283.349,A -85,B 0,C 180,E1 -6312.035,E2 -6312.035} C_VEL
LIN {X 0,Y 495.815,Z 283.352,A -85,B 0,C 180,E1 -6315.452,E2 -6315.452} C_VEL
LIN {X 0,Y 495.799,Z 283.353,A -85,B 0,C 180,E1 -6318.248,E2 -6318.248} C_VEL
LIN {X 0,Y 495.766,Z 283.354,A -85,B 0,C 180,E1 -6320.757,E2 -6320.757} C_VEL
LIN {X 0,Y 495.744,Z 283.358,A -85,B 0,C 180,E1 -6323.388,E2 -6323.388} C_VEL
LIN {X 0,Y 495.784,Z 283.356,A -85,B 0,C 180,E1 -6326.068,E2 -6326.068} C_VEL
LIN {X 0,Y 495.762,Z 283.356,A -85,B 0,C 180,E1 -6328.816,E2 -6328.816} C_VEL
LIN {X 0,Y 495.752,Z 283.355,A -85,B 0,C 180,E1 -6331.727,E2 -6331.727} C_VEL
LIN {X 0,Y 495.76,Z 283.354,A -85,B 0,C 180,E1 -6334.694,E2 -6334.694} C_VEL
LIN {X 0,Y 495.723,Z 283.36,A -85,B 0,C 180,E1 -6337.562,E2 -6337.562} C_VEL
LIN {X 0,Y 495.761,Z 283.356,A -85,B 0,C 180,E1 -6340.701,E2 -6340.701} C_VEL
LIN {X 0,Y 495.729,Z 283.36,A -85,B 0,C 180,E1 -6344.002,E2 -6344.002} C_VEL
LIN {X 0,Y 495.694,Z 283.367,A -85,B 0,C 180,E1 -6347.115,E2 -6347.115} C_VEL
LIN {X 0,Y 495.958,Z 286.35,A -85,B 0,C 180,E1 -6349.32,E2 -6349.32} C_VEL
LIN {X 0,Y 495.844,Z 290.954,A -85,B 0,C 180,E1 -6352.536,E2 -6352.536} C_VEL
LIN {X 0,Y 495.752,Z 295.296,A -85,B 0,C 180,E1 -6355.456,E2 -6355.456} C_VEL
LIN {X 0,Y 495.58,Z 299.752,A -85,B 0,C 180,E1 -6358.352,E2 -6358.352} C_VEL
LIN {X 0,Y 495.501,Z 303.111,A -85,B 0,C 180,E1 -6360.486,E2 -6360.486} C_VEL
LIN {X 0,Y 494.779,Z 304.248,A -85,B 0,C 180,E1 -6361.151,E2 -6361.151} C_VEL
LIN {X 0,Y 491.873,Z 306.281,A -85,B 0,C 180,E1 -6362.227,E2 -6362.227} C_VEL
LIN {X 0,Y 489.434,Z 307.93,A -85,B 0,C 180,E1 -6363.093,E2 -6363.093} C_VEL
LIN {X 0,Y 488.377,Z 309.125,A -85,B 0,C 180,E1 -6363.764,E2 -6363.764} C_VEL
LIN {X 0,Y 488.284,Z 309.504,A -85,B 0,C 180,E1 -6363.992,E2 -6363.992} C_VEL
LIN {X 0,Y 488.218,Z 313.19,A -85,B 0,C 180,E1 -6366.231,E2 -6366.231} C_VEL
LIN {X 0,Y 488.125,Z 318.255,A -85,B 0,C 180,E1 -6369.25,E2 -6369.25} C_VEL
LIN {X 0,Y 492.616,Z 334.754,A -85,B 0,C 180,E1 -6369.798,E2 -6369.798} C_VEL
LIN {X 0,Y 493.85,Z 340.763,A -85,B 0,C 180,E1 -6370.03,E2 -6370.03} C_VEL
LIN {X 0,Y 493.382,Z 355.047,A -85,B 0,C 180,E1 -6370.544,E2 -6370.544} C_VEL
LIN {X 0,Y 492.746,Z 368.445,A -85,B 0,C 180,E1 -6371.174,E2 -6371.174} C_VEL
LIN {X 0,Y 492.095,Z 382.469,A -85,B 0,C 180,E1 -6372.011,E2 -6372.011} C_VEL
LIN {X 0,Y 491.413,Z 395.286,A -85,B 0,C 180,E1 -6372.952,E2 -6372.952} C_VEL
LIN {X 0,Y 490.696,Z 407.867,A -85,B 0,C 180,E1 -6374.07,E2 -6374.07} C_VEL
LIN {X 0,Y 490.081,Z 418.989,A -85,B 0,C 180,E1 -6375.254,E2 -6375.254} C_VEL
LIN {X 0,Y 489.516,Z 428.968,A -85,B 0,C 180,E1 -6376.509,E2 -6376.509} C_VEL
LIN {X 0,Y 488.961,Z 438.6,A -85,B 0,C 180,E1 -6377.951,E2 -6377.951} C_VEL
LIN {X 0,Y 488.638,Z 446.839,A -85,B 0,C 180,E1 -6379.434,E2 -6379.434} C_VEL
LIN {X 0,Y 488.322,Z 453.543,A -85,B 0,C 180,E1 -6380.891,E2 -6380.891} C_VEL
LIN {X 0,Y 488.122,Z 459.756,A -85,B 0,C 180,E1 -6382.555,E2 -6382.555} C_VEL
LIN {X 0,Y 488.043,Z 464.556,A -85,B 0,C 180,E1 -6384.215,E2 -6384.215} C_VEL
LIN {X 0,Y 487.899,Z 468.076,A -85,B 0,C 180,E1 -6385.87,E2 -6385.87} C_VEL
LIN {X 0,Y 487.905,Z 470.406,A -85,B 0,C 180,E1 -6387.524,E2 -6387.524} C_VEL
LIN {X 0,Y 487.83,Z 471.6,A -85,B 0,C 180,E1 -6389.175,E2 -6389.175} C_VEL
LIN {X 0,Y 487.831,Z 471.618,A -85,B 0,C 180,E1 -6390.826,E2 -6390.826} C_VEL
LIN {X 0,Y 487.906,Z 470.497,A -85,B 0,C 180,E1 -6392.477,E2 -6392.477} C_VEL
LIN {X 0,Y 487.898,Z 468.237,A -85,B 0,C 180,E1 -6394.13,E2 -6394.13} C_VEL
LIN {X 0,Y 488.028,Z 464.784,A -85,B 0,C 180,E1 -6395.786,E2 -6395.786} C_VEL
LIN {X 0,Y 488.119,Z 460.057,A -85,B 0,C 180,E1 -6397.446,E2 -6397.446} C_VEL
LIN {X 0,Y 488.313,Z 453.933,A -85,B 0,C 180,E1 -6399.109,E2 -6399.109} C_VEL
LIN {X 0,Y 488.722,Z 446.222,A -85,B 0,C 180,E1 -6400.775,E2 -6400.775} C_VEL
LIN {X 0,Y 489.023,Z 437.988,A -85,B 0,C 180,E1 -6402.241,E2 -6402.241} C_VEL
LIN {X 0,Y 489.562,Z 428.105,A -85,B 0,C 180,E1 -6403.702,E2 -6403.702} C_VEL
LIN {X 0,Y 490.108,Z 417.958,A -85,B 0,C 180,E1 -6404.958,E2 -6404.958} C_VEL
LIN {X 0,Y 490.726,Z 407.608,A -85,B 0,C 180,E1 -6406.044,E2 -6406.044} C_VEL
LIN {X 0,Y 491.417,Z 395.065,A -85,B 0,C 180,E1 -6407.156,E2 -6407.156} C_VEL
LIN {X 0,Y 492.116,Z 382.206,A -85,B 0,C 180,E1 -6408.096,E2 -6408.096} C_VEL
LIN {X 0,Y 492.703,Z 370.093,A -85,B 0,C 180,E1 -6408.828,E2 -6408.828} C_VEL
LIN {X 0,Y 493.345,Z 355.794,A -85,B 0,C 180,E1 -6409.516,E2 -6409.516} C_VEL
LIN {X 0,Y 493.796,Z 341.474,A -85,B 0,C 180,E1 -6410.041,E2 -6410.041} C_VEL
LIN {X 0,Y 493.559,Z 338.831,A -85,B 0,C 180,E1 -6410.13,E2 -6410.13} C_VEL
LIN {X 0,Y 489.853,Z 324.505,A -85,B 0,C 180,E1 -6410.648,E2 -6410.648} C_VEL
LIN {X 0,Y 488.141,Z 318.264,A -85,B 0,C 180,E1 -6410.845,E2 -6410.845} C_VEL
LIN {X 0,Y 488.217,Z 313.384,A -85,B 0,C 180,E1 -6413.77,E2 -6413.77} C_VEL
LIN {X 0,Y 488.331,Z 308.378,A -85,B 0,C 180,E1 -6416.837,E2 -6416.837} C_VEL
LIN {X 0,Y 488.439,Z 304.465,A -85,B 0,C 180,E1 -6419.289,E2 -6419.289} C_VEL
LIN {X 0,Y 488.566,Z 299.983,A -85,B 0,C 180,E1 -6422.157,E2 -6422.157} C_VEL
LIN {X 0,Y 488.727,Z 295.494,A -85,B 0,C 180,E1 -6425.114,E2 -6425.114} C_VEL
LIN {X 0,Y 488.807,Z 291.004,A -85,B 0,C 180,E1 -6428.188,E2 -6428.188} C_VEL
LIN {X 0,Y 488.948,Z 287.903,A -85,B 0,C 180,E1 -6430.376,E2 -6430.376} C_VEL
LIN {X 0,Y 488.723,Z 284.6,A -85,B 0,C 180,E1 -6432.828,E2 -6432.828} C_VEL
LIN {X 0,Y 488.694,Z 284.24,A -85,B 0,C 180,E1 -6434.023,E2 -6434.023} C_VEL
LIN {X 0,Y 488.708,Z 284.239,A -85,B 0,C 180,E1 -6437.173,E2 -6437.173} C_VEL
LIN {X 0,Y 488.732,Z 284.23,A -85,B 0,C 180,E1 -6439.676,E2 -6439.676} C_VEL
LIN {X 0,Y 488.677,Z 284.24,A -85,B 0,C 180,E1 -6442.841,E2 -6442.841} C_VEL
LIN {X 0,Y 488.727,Z 284.233,A -85,B 0,C 180,E1 -6445.887,E2 -6445.887} C_VEL
LIN {X 0,Y 488.689,Z 284.237,A -85,B 0,C 180,E1 -6448.82,E2 -6448.82} C_VEL
LIN {X 0,Y 488.709,Z 284.233,A -85,B 0,C 180,E1 -6451.669,E2 -6451.669} C_VEL
LIN {X 0,Y 488.711,Z 284.234,A -85,B 0,C 180,E1 -6454.442,E2 -6454.442} C_VEL
LIN {X 0,Y 488.721,Z 284.235,A -85,B 0,C 180,E1 -6457.153,E2 -6457.153} C_VEL
LIN {X 0,Y 488.721,Z 284.233,A -85,B 0,C 180,E1 -6459.81,E2 -6459.81} C_VEL
LIN {X 0,Y 488.73,Z 284.231,A -85,B 0,C 180,E1 -6462.423,E2 -6462.423} C_VEL
LIN {X 0,Y 488.756,Z 284.23,A -85,B 0,C 180,E1 -6464.999,E2 -6464.999} C_VEL
LIN {X 0,Y 488.802,Z 284.222,A -85,B 0,C 180,E1 -6468.387,E2 -6468.387} C_VEL
LIN {X 0,Y 488.783,Z 284.223,A -85,B 0,C 180,E1 -6471.733,E2 -6471.733} C_VEL
LIN {X 0,Y 488.833,Z 284.22,A -85,B 0,C 180,E1 -6474.224,E2 -6474.224} C_VEL
LIN {X 0,Y 488.959,Z 284.202,A -85,B 0,C 180,E1 -6477.529,E2 -6477.529} C_VEL
LIN {X 0,Y 488.964,Z 284.206,A -85,B 0,C 180,E1 -6480,E2 -6480} C_VEL
LIN {X 0,Y 488.959,Z 284.202,A -85,B 0,C 180,E1 -6482.471,E2 -6482.471} C_VEL
LIN {X 0,Y 488.834,Z 284.219,A -85,B 0,C 180,E1 -6485.776,E2 -6485.776} C_VEL
LIN {X 0,Y 488.783,Z 284.224,A -85,B 0,C 180,E1 -6488.267,E2 -6488.267} C_VEL
LIN {X 0,Y 488.802,Z 284.222,A -85,B 0,C 180,E1 -6491.612,E2 -6491.612} C_VEL
LIN {X 0,Y 488.757,Z 284.229,A -85,B 0,C 180,E1 -6495,E2 -6495} C_VEL
LIN {X 0,Y 488.752,Z 284.233,A -85,B 0,C 180,E1 -6498.442,E2 -6498.442} C_VEL
LIN {X 0,Y 488.702,Z 284.235,A -85,B 0,C 180,E1 -6501.071,E2 -6501.071} C_VEL
LIN {X 0,Y 488.685,Z 284.236,A -85,B 0,C 180,E1 -6503.746,E2 -6503.746} C_VEL
LIN {X 0,Y 488.787,Z 284.224,A -85,B 0,C 180,E1 -6506.943,E2 -6506.943} C_VEL
LIN {X 0,Y 488.705,Z 284.238,A -85,B 0,C 180,E1 -6510.363,E2 -6510.363} C_VEL
LIN {X 0,Y 488.731,Z 284.237,A -85,B 0,C 180,E1 -6513.484,E2 -6513.484} C_VEL
LIN {X 0,Y 488.678,Z 284.242,A -85,B 0,C 180,E1 -6516.354,E2 -6516.354} C_VEL
LIN {X 0,Y 488.699,Z 284.238,A -85,B 0,C 180,E1 -6519.254,E2 -6519.254} C_VEL
LIN {X 0,Y 488.685,Z 284.24,A -85,B 0,C 180,E1 -6522.526,E2 -6522.526} C_VEL
LIN {X 0,Y 488.747,Z 284.294,A -85,B 0,C 180,E1 -6525.758,E2 -6525.758} C_VEL
LIN {X 0,Y 489.226,Z 288.231,A -85,B 0,C 180,E1 -6528.332,E2 -6528.332} C_VEL
LIN {X 0,Y 489.183,Z 292.4,A -85,B 0,C 180,E1 -6530.878,E2 -6530.878} C_VEL
LIN {X 0,Y 489.006,Z 297.558,A -85,B 0,C 180,E1 -6533.896,E2 -6533.896} C_VEL
LIN {X 0,Y 488.789,Z 302.857,A -85,B 0,C 180,E1 -6536.881,E2 -6536.881} C_VEL
LIN {X 0,Y 488.643,Z 308.165,A -85,B 0,C 180,E1 -6539.775,E2 -6539.775} C_VEL
LIN {X 0,Y 488.437,Z 313.485,A -85,B 0,C 180,E1 -6542.585,E2 -6542.585} C_VEL
LIN {X 0,Y 488.347,Z 318.817,A -85,B 0,C 180,E1 -6545.333,E2 -6545.333} C_VEL
LIN {X 0,Y 488.201,Z 324.154,A -85,B 0,C 180,E1 -6548.02,E2 -6548.02} C_VEL
LIN {X 0,Y 488.174,Z 326.517,A -85,B 0,C 180,E1 -6549.194,E2 -6549.194} C_VEL
LIN {X 0,Y 492.54,Z 343.644,A -85,B 0,C 180,E1 -6549.748,E2 -6549.748} C_VEL
LIN {X 0,Y 493.75,Z 349.495,A -85,B 0,C 180,E1 -6549.972,E2 -6549.972} C_VEL
LIN {X 0,Y 493.369,Z 363.215,A -85,B 0,C 180,E1 -6550.463,E2 -6550.463} C_VEL
LIN {X 0,Y 492.72,Z 376.343,A -85,B 0,C 180,E1 -6551.065,E2 -6551.065} C_VEL
LIN {X 0,Y 492.036,Z 390.641,A -85,B 0,C 180,E1 -6551.901,E2 -6551.901} C_VEL
LIN {X 0,Y 491.352,Z 403.654,A -85,B 0,C 180,E1 -6552.842,E2 -6552.842} C_VEL
LIN {X 0,Y 490.656,Z 416.351,A -85,B 0,C 180,E1 -6553.956,E2 -6553.956} C_VEL
LIN {X 0,Y 490.037,Z 426.789,A -85,B 0,C 180,E1 -6555.039,E2 -6555.039} C_VEL
LIN {X 0,Y 489.515,Z 437.019,A -85,B 0,C 180,E1 -6556.297,E2 -6556.297} C_VEL
LIN {X 0,Y 488.899,Z 447.428,A -85,B 0,C 180,E1 -6557.825,E2 -6557.825} C_VEL
LIN {X 0,Y 488.639,Z 455.318,A -85,B 0,C 180,E1 -6559.223,E2 -6559.223} C_VEL
LIN {X 0,Y 488.274,Z 463.114,A -85,B 0,C 180,E1 -6560.89,E2 -6560.89} C_VEL
LIN {X 0,Y 488.075,Z 469.315,A -85,B 0,C 180,E1 -6562.554,E2 -6562.554} C_VEL
LIN {X 0,Y 488.001,Z 474.11,A -85,B 0,C 180,E1 -6564.214,E2 -6564.214} C_VEL
LIN {X 0,Y 487.89,Z 477.622,A -85,B 0,C 180,E1 -6565.869,E2 -6565.869} C_VEL
LIN {X 0,Y 487.883,Z 479.932,A -85,B 0,C 180,E1 -6567.523,E2 -6567.523} C_VEL
LIN {X 0,Y 487.83,Z 481.094,A -85,B 0,C 180,E1 -6569.174,E2 -6569.174} C_VEL
LIN {X 0,Y 487.83,Z 481.094,A -85,B 0,C 180,E1 -6570.825,E2 -6570.825} C_VEL
LIN {X 0,Y 487.883,Z 479.928,A -85,B 0,C 180,E1 -6572.476,E2 -6572.476} C_VEL
LIN {X 0,Y 487.89,Z 477.618,A -85,B 0,C 180,E1 -6574.13,E2 -6574.13} C_VEL
LIN {X 0,Y 488.01,Z 474.113,A -85,B 0,C 180,E1 -6575.785,E2 -6575.785} C_VEL
LIN {X 0,Y 488.075,Z 469.321,A -85,B 0,C 180,E1 -6577.446,E2 -6577.446} C_VEL
LIN {X 0,Y 488.274,Z 463.113,A -85,B 0,C 180,E1 -6579.109,E2 -6579.109} C_VEL
LIN {X 0,Y 488.636,Z 455.315,A -85,B 0,C 180,E1 -6580.776,E2 -6580.776} C_VEL
LIN {X 0,Y 488.962,Z 447.212,A -85,B 0,C 180,E1 -6582.209,E2 -6582.209} C_VEL
LIN {X 0,Y 489.515,Z 437.024,A -85,B 0,C 180,E1 -6583.703,E2 -6583.703} C_VEL
LIN {X 0,Y 490.049,Z 426.795,A -85,B 0,C 180,E1 -6584.959,E2 -6584.959} C_VEL
LIN {X 0,Y 490.762,Z 414.499,A -85,B 0,C 180,E1 -6586.226,E2 -6586.226} C_VEL
LIN {X 0,Y 491.503,Z 401.044,A -85,B 0,C 180,E1 -6587.366,E2 -6587.366} C_VEL
LIN {X 0,Y 492.223,Z 387.439,A -85,B 0,C 180,E1 -6588.307,E2 -6588.307} C_VEL
LIN {X 0,Y 492.923,Z 373.346,A -85,B 0,C 180,E1 -6589.088,E2 -6589.088} C_VEL
LIN {X 0,Y 493.461,Z 358.407,A -85,B 0,C 180,E1 -6589.732,E2 -6589.732} C_VEL
LIN {X 0,Y 493.617,Z 348.296,A -85,B 0,C 180,E1 -6590.069,E2 -6590.069} C_VEL
LIN {X 0,Y 489.802,Z 332.84,A -85,B 0,C 180,E1 -6590.616,E2 -6590.616} C_VEL
LIN {X 0,Y 488.177,Z 326.494,A -85,B 0,C 180,E1 -6590.826,E2 -6590.826} C_VEL
LIN {X 0,Y 488.266,Z 320.642,A -85,B 0,C 180,E1 -6593.767,E2 -6593.767} C_VEL
LIN {X 0,Y 488.416,Z 314.635,A -85,B 0,C 180,E1 -6596.857,E2 -6596.857} C_VEL
LIN {X 0,Y 488.657,Z 308.219,A -85,B 0,C 180,E1 -6600.223,E2 -6600.223} C_VEL
LIN {X 0,Y 488.823,Z 302.185,A -85,B 0,C 180,E1 -6603.5,E2 -6603.5} C_VEL
LIN {X 0,Y 489.028,Z 297.019,A -85,B 0,C 180,E1 -6606.41,E2 -6606.41} C_VEL
LIN {X 0,Y 489.184,Z 292.249,A -85,B 0,C 180,E1 -6609.207,E2 -6609.207} C_VEL
LIN {X 0,Y 489.197,Z 288.224,A -85,B 0,C 180,E1 -6611.664,E2 -6611.664} C_VEL
LIN {X 0,Y 488.752,Z 284.228,A -85,B 0,C 180,E1 -6614.29,E2 -6614.29} C_VEL
LIN {X 0,Y 488.685,Z 284.241,A -85,B 0,C 180,E1 -6617.474,E2 -6617.474} C_VEL
LIN {X 0,Y 488.726,Z 284.233,A -85,B 0,C 180,E1 -6619.676,E2 -6619.676} C_VEL
LIN {X 0,Y 488.672,Z 284.241,A -85,B 0,C 180,E1 -6622.84,E2 -6622.84} C_VEL
LIN {X 0,Y 488.722,Z 284.235,A -85,B 0,C 180,E1 -6625.887,E2 -6625.887} C_VEL
LIN {X 0,Y 488.687,Z 284.239,A -85,B 0,C 180,E1 -6628.82,E2 -6628.82} C_VEL
LIN {X 0,Y 488.734,Z 284.232,A -85,B 0,C 180,E1 -6631.671,E2 -6631.671} C_VEL
LIN {X 0,Y 488.74,Z 284.231,A -85,B 0,C 180,E1 -6634.444,E2 -6634.444} C_VEL
LIN {X 0,Y 488.716,Z 284.237,A -85,B 0,C 180,E1 -6637.153,E2 -6637.153} C_VEL
LIN {X 0,Y 488.717,Z 284.235,A -85,B 0,C 180,E1 -6639.81,E2 -6639.81} C_VEL
LIN {X 0,Y 488.725,Z 284.231,A -85,B 0,C 180,E1 -6642.423,E2 -6642.423} C_VEL
LIN {X 0,Y 488.752,Z 284.229,A -85,B 0,C 180,E1 -6644.999,E2 -6644.999} C_VEL
LIN {X 0,Y 488.8,Z 284.221,A -85,B 0,C 180,E1 -6648.388,E2 -6648.388} C_VEL
LIN {X 0,Y 488.779,Z 284.224,A -85,B 0,C 180,E1 -6651.733,E2 -6651.733} C_VEL
LIN {X 0,Y 488.83,Z 284.218,A -85,B 0,C 180,E1 -6654.224,E2 -6654.224} C_VEL
LIN {X 0,Y 488.955,Z 284.201,A -85,B 0,C 180,E1 -6657.529,E2 -6657.529} C_VEL
LIN {X 0,Y 488.904,Z 284.209,A -85,B 0,C 180,E1 -6660.824,E2 -6660.824} C_VEL
LIN {X 0,Y 488.955,Z 284.203,A -85,B 0,C 180,E1 -6662.471,E2 -6662.471} C_VEL
LIN {X 0,Y 488.83,Z 284.22,A -85,B 0,C 180,E1 -6665.776,E2 -6665.776} C_VEL
LIN {X 0,Y 488.778,Z 284.223,A -85,B 0,C 180,E1 -6668.267,E2 -6668.267} C_VEL
LIN {X 0,Y 488.797,Z 284.221,A -85,B 0,C 180,E1 -6671.613,E2 -6671.613} C_VEL
LIN {X 0,Y 488.752,Z 284.229,A -85,B 0,C 180,E1 -6675.001,E2 -6675.001} C_VEL
LIN {X 0,Y 488.747,Z 284.233,A -85,B 0,C 180,E1 -6678.443,E2 -6678.443} C_VEL
LIN {X 0,Y 488.699,Z 284.235,A -85,B 0,C 180,E1 -6681.071,E2 -6681.071} C_VEL
LIN {X 0,Y 488.685,Z 284.236,A -85,B 0,C 180,E1 -6683.746,E2 -6683.746} C_VEL
LIN {X 0,Y 488.783,Z 284.223,A -85,B 0,C 180,E1 -6686.944,E2 -6686.944} C_VEL
LIN {X 0,Y 488.703,Z 284.235,A -85,B 0,C 180,E1 -6690.364,E2 -6690.364} C_VEL
LIN {X 0,Y 488.728,Z 284.232,A -85,B 0,C 180,E1 -6693.485,E2 -6693.485} C_VEL
LIN {X 0,Y 488.674,Z 284.238,A -85,B 0,C 180,E1 -6696.355,E2 -6696.355} C_VEL
LIN {X 0,Y 488.696,Z 284.236,A -85,B 0,C 180,E1 -6699.255,E2 -6699.255} C_VEL
LIN {X 0,Y 488.702,Z 284.238,A -85,B 0,C 180,E1 -6701.601,E2 -6701.601} C_VEL
LIN {X 0,Y 488.707,Z 284.235,A -85,B 0,C 180,E1 -6704.802,E2 -6704.802} C_VEL
LIN {X 0,Y 488.692,Z 284.48,A -85,B 0,C 180,E1 -6707.176,E2 -6707.176} C_VEL
LIN {X 0,Y 488.932,Z 287.878,A -85,B 0,C 180,E1 -6709.698,E2 -6709.698} C_VEL
LIN {X 0,Y 488.776,Z 292.359,A -85,B 0,C 180,E1 -6712.851,E2 -6712.851} C_VEL
LIN {X 0,Y 488.675,Z 296.825,A -85,B 0,C 180,E1 -6715.884,E2 -6715.884} C_VEL
LIN {X 0,Y 488.504,Z 301.284,A -85,B 0,C 180,E1 -6718.808,E2 -6718.808} C_VEL
LIN {X 0,Y 488.411,Z 305.731,A -85,B 0,C 180,E1 -6721.651,E2 -6721.651} C_VEL
LIN {X 0,Y 488.284,Z 309.504,A -85,B 0,C 180,E1 -6723.992,E2 -6723.992} C_VEL
LIN {X 0,Y 487.592,Z 310.675,A -85,B 0,C 180,E1 -6724.666,E2 -6724.666} C_VEL
LIN {X 0,Y 484.697,Z 312.745,A -85,B 0,C 180,E1 -6725.755,E2 -6725.755} C_VEL
LIN {X 0,Y 482.249,Z 314.418,A -85,B 0,C 180,E1 -6726.633,E2 -6726.633} C_VEL
LIN {X 0,Y 481.184,Z 315.634,A -85,B 0,C 180,E1 -6727.313,E2 -6727.313} C_VEL
LIN {X 0,Y 481.089,Z 316.023,A -85,B 0,C 180,E1 -6727.544,E2 -6727.544} C_VEL
LIN {X 0,Y 481.045,Z 318.318,A -85,B 0,C 180,E1 -6728.927,E2 -6728.927} C_VEL
LIN {X 0,Y 485.698,Z 335.204,A -85,B 0,C 180,E1 -6729.509,E2 -6729.509} C_VEL
LIN {X 0,Y 487.165,Z 341.848,A -85,B 0,C 180,E1 -6729.774,E2 -6729.774} C_VEL
LIN {X 0,Y 486.655,Z 356.801,A -85,B 0,C 180,E1 -6730.335,E2 -6730.335} C_VEL
LIN {X 0,Y 485.934,Z 370.508,A -85,B 0,C 180,E1 -6731.01,E2 -6731.01} C_VEL
LIN {X 0,Y 485.235,Z 384.128,A -85,B 0,C 180,E1 -6731.857,E2 -6731.857} C_VEL
LIN {X 0,Y 484.525,Z 396.653,A -85,B 0,C 180,E1 -6732.811,E2 -6732.811} C_VEL
LIN {X 0,Y 483.824,Z 408.103,A -85,B 0,C 180,E1 -6733.854,E2 -6733.854} C_VEL
LIN {X 0,Y 483.18,Z 419.064,A -85,B 0,C 180,E1 -6735.039,E2 -6735.039} C_VEL
LIN {X 0,Y 482.559,Z 429.042,A -85,B 0,C 180,E1 -6736.311,E2 -6736.311} C_VEL
LIN {X 0,Y 482.044,Z 437.894,A -85,B 0,C 180,E1 -6737.643,E2 -6737.643} C_VEL
LIN {X 0,Y 481.639,Z 446.911,A -85,B 0,C 180,E1 -6739.278,E2 -6739.278} C_VEL
LIN {X 0,Y 481.268,Z 453.616,A -85,B 0,C 180,E1 -6740.757,E2 -6740.757} C_VEL
LIN {X 0,Y 481.042,Z 459.827,A -85,B 0,C 180,E1 -6742.445,E2 -6742.445} C_VEL
LIN {X 0,Y 480.964,Z 464.627,A -85,B 0,C 180,E1 -6744.13,E2 -6744.13} C_VEL
LIN {X 0,Y 480.802,Z 468.147,A -85,B 0,C 180,E1 -6745.809,E2 -6745.809} C_VEL
LIN {X 0,Y 480.819,Z 470.476,A -85,B 0,C 180,E1 -6747.487,E2 -6747.487} C_VEL
LIN {X 0,Y 480.757,Z 471.669,A -85,B 0,C 180,E1 -6749.163,E2 -6749.163} C_VEL
LIN {X 0,Y 480.757,Z 471.686,A -85,B 0,C 180,E1 -6750.838,E2 -6750.838} C_VEL
LIN {X 0,Y 480.82,Z 470.565,A -85,B 0,C 180,E1 -6752.514,E2 -6752.514} C_VEL
LIN {X 0,Y 480.801,Z 468.305,A -85,B 0,C 180,E1 -6754.192,E2 -6754.192} C_VEL
LIN {X 0,Y 480.93,Z 464.851,A -85,B 0,C 180,E1 -6755.871,E2 -6755.871} C_VEL
LIN {X 0,Y 481.036,Z 460.124,A -85,B 0,C 180,E1 -6757.556,E2 -6757.556} C_VEL
LIN {X 0,Y 481.258,Z 453.999,A -85,B 0,C 180,E1 -6759.244,E2 -6759.244} C_VEL
LIN {X 0,Y 481.695,Z 446.288,A -85,B 0,C 180,E1 -6760.934,E2 -6760.934} C_VEL
LIN {X 0,Y 481.996,Z 438.586,A -85,B 0,C 180,E1 -6762.331,E2 -6762.331} C_VEL
LIN {X 0,Y 482.604,Z 428.17,A -85,B 0,C 180,E1 -6763.903,E2 -6763.903} C_VEL
LIN {X 0,Y 483.191,Z 418.022,A -85,B 0,C 180,E1 -6765.178,E2 -6765.178} C_VEL
LIN {X 0,Y 483.921,Z 406.449,A -85,B 0,C 180,E1 -6766.4,E2 -6766.4} C_VEL
LIN {X 0,Y 484.675,Z 393.837,A -85,B 0,C 180,E1 -6767.511,E2 -6767.511} C_VEL
LIN {X 0,Y 485.419,Z 380.687,A -85,B 0,C 180,E1 -6768.464,E2 -6768.464} C_VEL
LIN {X 0,Y 486.109,Z 368.164,A -85,B 0,C 180,E1 -6769.203,E2 -6769.203} C_VEL
LIN {X 0,Y 486.695,Z 353.443,A -85,B 0,C 180,E1 -6769.895,E2 -6769.895} C_VEL
LIN {X 0,Y 487.047,Z 340.831,A -85,B 0,C 180,E1 -6770.352,E2 -6770.352} C_VEL
LIN {X 0,Y 483.292,Z 326.182,A -85,B 0,C 180,E1 -6770.911,E2 -6770.911} C_VEL
LIN {X 0,Y 481.041,Z 318.346,A -85,B 0,C 180,E1 -6771.159,E2 -6771.159} C_VEL
LIN {X 0,Y 481.177,Z 313.451,A -85,B 0,C 180,E1 -6774.14,E2 -6774.14} C_VEL
LIN {X 0,Y 481.27,Z 308.809,A -85,B 0,C 180,E1 -6777.028,E2 -6777.028} C_VEL
LIN {X 0,Y 481.408,Z 304.51,A -85,B 0,C 180,E1 -6779.759,E2 -6779.759} C_VEL
LIN {X 0,Y 481.526,Z 300.033,A -85,B 0,C 180,E1 -6782.685,E2 -6782.685} C_VEL
LIN {X 0,Y 481.68,Z 296.265,A -85,B 0,C 180,E1 -6785.207,E2 -6785.207} C_VEL
LIN {X 0,Y 481.77,Z 292.196,A -85,B 0,C 180,E1 -6788.025,E2 -6788.025} C_VEL
LIN {X 0,Y 481.899,Z 288.502,A -85,B 0,C 180,E1 -6790.679,E2 -6790.679} C_VEL
LIN {X 0,Y 481.639,Z 285.118,A -85,B 0,C 180,E1 -6793.299,E2 -6793.299} C_VEL
LIN {X 0,Y 481.657,Z 285.117,A -85,B 0,C 180,E1 -6795.641,E2 -6795.641} C_VEL
LIN {X 0,Y 481.655,Z 285.115,A -85,B 0,C 180,E1 -6798.958,E2 -6798.958} C_VEL
LIN {X 0,Y 481.653,Z 285.117,A -85,B 0,C 180,E1 -6801.992,E2 -6801.992} C_VEL
LIN {X 0,Y 481.685,Z 285.111,A -85,B 0,C 180,E1 -6805.317,E2 -6805.317} C_VEL
LIN {X 0,Y 481.642,Z 285.116,A -85,B 0,C 180,E1 -6808.311,E2 -6808.311} C_VEL
LIN {X 0,Y 481.671,Z 285.113,A -85,B 0,C 180,E1 -6811.217,E2 -6811.217} C_VEL
LIN {X 0,Y 481.666,Z 285.115,A -85,B 0,C 180,E1 -6814.041,E2 -6814.041} C_VEL
LIN {X 0,Y 481.671,Z 285.112,A -85,B 0,C 180,E1 -6816.812,E2 -6816.812} C_VEL
LIN {X 0,Y 481.692,Z 285.108,A -85,B 0,C 180,E1 -6819.502,E2 -6819.502} C_VEL
LIN {X 0,Y 481.704,Z 285.107,A -85,B 0,C 180,E1 -6822.158,E2 -6822.158} C_VEL
LIN {X 0,Y 481.738,Z 285.106,A -85,B 0,C 180,E1 -6824.776,E2 -6824.776} C_VEL
LIN {X 0,Y 481.747,Z 285.102,A -85,B 0,C 180,E1 -6828.215,E2 -6828.215} C_VEL
LIN {X 0,Y 481.738,Z 285.101,A -85,B 0,C 180,E1 -6831.611,E2 -6831.611} C_VEL
LIN {X 0,Y 481.792,Z 285.098,A -85,B 0,C 180,E1 -6834.139,E2 -6834.139} C_VEL
LIN {X 0,Y 481.926,Z 285.079,A -85,B 0,C 180,E1 -6837.492,E2 -6837.492} C_VEL
LIN {X 0,Y 481.935,Z 285.081,A -85,B 0,C 180,E1 -6840,E2 -6840} C_VEL
LIN {X 0,Y 481.926,Z 285.079,A -85,B 0,C 180,E1 -6842.507,E2 -6842.507} C_VEL
LIN {X 0,Y 481.792,Z 285.097,A -85,B 0,C 180,E1 -6845.861,E2 -6845.861} C_VEL
LIN {X 0,Y 481.738,Z 285.102,A -85,B 0,C 180,E1 -6848.389,E2 -6848.389} C_VEL
LIN {X 0,Y 481.747,Z 285.102,A -85,B 0,C 180,E1 -6851.785,E2 -6851.785} C_VEL
LIN {X 0,Y 481.738,Z 285.106,A -85,B 0,C 180,E1 -6855.224,E2 -6855.224} C_VEL
LIN {X 0,Y 481.708,Z 285.107,A -85,B 0,C 180,E1 -6858.722,E2 -6858.722} C_VEL
LIN {X 0,Y 481.641,Z 285.118,A -85,B 0,C 180,E1 -6861.395,E2 -6861.395} C_VEL
LIN {X 0,Y 481.67,Z 285.111,A -85,B 0,C 180,E1 -6864.113,E2 -6864.113} C_VEL
LIN {X 0,Y 481.742,Z 285.103,A -85,B 0,C 180,E1 -6867.139,E2 -6867.139} C_VEL
LIN {X 0,Y 481.674,Z 285.112,A -85,B 0,C 180,E1 -6869.741,E2 -6869.741} C_VEL
LIN {X 0,Y 481.668,Z 285.115,A -85,B 0,C 180,E1 -6872.674,E2 -6872.674} C_VEL
LIN {X 0,Y 481.632,Z 285.119,A -85,B 0,C 180,E1 -6875.71,E2 -6875.71} C_VEL
LIN {X 0,Y 481.669,Z 285.114,A -85,B 0,C 180,E1 -6878.859,E2 -6878.859} C_VEL
LIN {X 0,Y 481.644,Z 285.116,A -85,B 0,C 180,E1 -6881.912,E2 -6881.912} C_VEL
LIN {X 0,Y 481.698,Z 285.18,A -85,B 0,C 180,E1 -6885.548,E2 -6885.548} C_VEL
LIN {X 0,Y 482.168,Z 288.893,A -85,B 0,C 180,E1 -6888.019,E2 -6888.019} C_VEL
LIN {X 0,Y 482.183,Z 292.217,A -85,B 0,C 180,E1 -6890.11,E2 -6890.11} C_VEL
LIN {X 0,Y 482.017,Z 297.563,A -85,B 0,C 180,E1 -6893.314,E2 -6893.314} C_VEL
LIN {X 0,Y 481.794,Z 302.807,A -85,B 0,C 180,E1 -6896.337,E2 -6896.337} C_VEL
LIN {X 0,Y 481.599,Z 308.37,A -85,B 0,C 180,E1 -6899.428,E2 -6899.428} C_VEL
LIN {X 0,Y 481.415,Z 313.436,A -85,B 0,C 180,E1 -6902.15,E2 -6902.15} C_VEL
LIN {X 0,Y 481.277,Z 318.757,A -85,B 0,C 180,E1 -6904.946,E2 -6904.946} C_VEL
LIN {X 0,Y 481.144,Z 324.089,A -85,B 0,C 180,E1 -6907.68,E2 -6907.68} C_VEL
LIN {X 0,Y 481.123,Z 326.45,A -85,B 0,C 180,E1 -6908.875,E2 -6908.875} C_VEL
LIN {X 0,Y 485.578,Z 343.625,A -85,B 0,C 180,E1 -6909.446,E2 -6909.446} C_VEL
LIN {X 0,Y 487.047,Z 351.149,A -85,B 0,C 180,E1 -6909.738,E2 -6909.738} C_VEL
LIN {X 0,Y 486.618,Z 364.782,A -85,B 0,C 180,E1 -6910.25,E2 -6910.25} C_VEL
LIN {X 0,Y 485.893,Z 378.264,A -85,B 0,C 180,E1 -6910.898,E2 -6910.898} C_VEL
LIN {X 0,Y 485.184,Z 392.155,A -85,B 0,C 180,E1 -6911.745,E2 -6911.745} C_VEL
LIN {X 0,Y 484.46,Z 404.877,A -85,B 0,C 180,E1 -6912.699,E2 -6912.699} C_VEL
LIN {X 0,Y 483.742,Z 417.028,A -85,B 0,C 180,E1 -6913.796,E2 -6913.796} C_VEL
LIN {X 0,Y 483.014,Z 428.505,A -85,B 0,C 180,E1 -6915.033,E2 -6915.033} C_VEL
LIN {X 0,Y 482.47,Z 438.464,A -85,B 0,C 180,E1 -6916.308,E2 -6916.308} C_VEL
LIN {X 0,Y 481.872,Z 447.886,A -85,B 0,C 180,E1 -6917.736,E2 -6917.736} C_VEL
LIN {X 0,Y 481.57,Z 456.331,A -85,B 0,C 180,E1 -6919.276,E2 -6919.276} C_VEL
LIN {X 0,Y 481.218,Z 463.044,A -85,B 0,C 180,E1 -6920.755,E2 -6920.755} C_VEL
LIN {X 0,Y 480.999,Z 469.245,A -85,B 0,C 180,E1 -6922.443,E2 -6922.443} C_VEL
LIN {X 0,Y 480.904,Z 474.04,A -85,B 0,C 180,E1 -6924.128,E2 -6924.128} C_VEL
LIN {X 0,Y 480.794,Z 477.552,A -85,B 0,C 180,E1 -6925.808,E2 -6925.808} C_VEL
LIN {X 0,Y 480.799,Z 479.863,A -85,B 0,C 180,E1 -6927.486,E2 -6927.486} C_VEL
LIN {X 0,Y 480.756,Z 481.026,A -85,B 0,C 180,E1 -6929.162,E2 -6929.162} C_VEL
LIN {X 0,Y 480.756,Z 481.025,A -85,B 0,C 180,E1 -6930.837,E2 -6930.837} C_VEL
LIN {X 0,Y 480.799,Z 479.859,A -85,B 0,C 180,E1 -6932.513,E2 -6932.513} C_VEL
LIN {X 0,Y 480.794,Z 477.549,A -85,B 0,C 180,E1 -6934.191,E2 -6934.191} C_VEL
LIN {X 0,Y 480.919,Z 474.043,A -85,B 0,C 180,E1 -6935.871,E2 -6935.871} C_VEL
LIN {X 0,Y 480.998,Z 469.251,A -85,B 0,C 180,E1 -6937.556,E2 -6937.556} C_VEL
LIN {X 0,Y 481.217,Z 463.044,A -85,B 0,C 180,E1 -6939.244,E2 -6939.244} C_VEL
LIN {X 0,Y 481.613,Z 455.246,A -85,B 0,C 180,E1 -6940.935,E2 -6940.935} C_VEL
LIN {X 0,Y 481.975,Z 446.699,A -85,B 0,C 180,E1 -6942.459,E2 -6942.459} C_VEL
LIN {X 0,Y 482.566,Z 436.954,A -85,B 0,C 180,E1 -6943.904,E2 -6943.904} C_VEL
LIN {X 0,Y 483.131,Z 426.726,A -85,B 0,C 180,E1 -6945.179,E2 -6945.179} C_VEL
LIN {X 0,Y 483.861,Z 415.109,A -85,B 0,C 180,E1 -6946.395,E2 -6946.395} C_VEL
LIN {X 0,Y 484.597,Z 402.306,A -85,B 0,C 180,E1 -6947.513,E2 -6947.513} C_VEL
LIN {X 0,Y 485.377,Z 388.992,A -85,B 0,C 180,E1 -6948.465,E2 -6948.465} C_VEL
LIN {X 0,Y 486.015,Z 376.282,A -85,B 0,C 180,E1 -6949.206,E2 -6949.206} C_VEL
LIN {X 0,Y 486.654,Z 362.036,A -85,B 0,C 180,E1 -6949.865,E2 -6949.865} C_VEL
LIN {X 0,Y 486.933,Z 349.658,A -85,B 0,C 180,E1 -6950.314,E2 -6950.314} C_VEL
LIN {X 0,Y 483.133,Z 334.104,A -85,B 0,C 180,E1 -6950.889,E2 -6950.889} C_VEL
LIN {X 0,Y 481.104,Z 326.469,A -85,B 0,C 180,E1 -6951.125,E2 -6951.125} C_VEL
LIN {X 0,Y 481.226,Z 320.581,A -85,B 0,C 180,E1 -6954.136,E2 -6954.136} C_VEL
LIN {X 0,Y 481.369,Z 315.014,A -85,B 0,C 180,E1 -6957.051,E2 -6957.051} C_VEL
LIN {X 0,Y 481.543,Z 309.947,A -85,B 0,C 180,E1 -6959.749,E2 -6959.749} C_VEL
LIN {X 0,Y 481.711,Z 304.607,A -85,B 0,C 180,E1 -6962.67,E2 -6962.67} C_VEL
LIN {X 0,Y 481.937,Z 299.284,A -85,B 0,C 180,E1 -6965.683,E2 -6965.683} C_VEL
LIN {X 0,Y 482.14,Z 293.977,A -85,B 0,C 180,E1 -6968.813,E2 -6968.813} C_VEL
LIN {X 0,Y 482.246,Z 290.438,A -85,B 0,C 180,E1 -6970.98,E2 -6970.98} C_VEL
LIN {X 0,Y 481.989,Z 286.915,A -85,B 0,C 180,E1 -6973.259,E2 -6973.259} C_VEL
LIN {X 0,Y 481.704,Z 285.107,A -85,B 0,C 180,E1 -6974.516,E2 -6974.516} C_VEL
LIN {X 0,Y 481.646,Z 285.116,A -85,B 0,C 180,E1 -6978.087,E2 -6978.087} C_VEL
LIN {X 0,Y 481.665,Z 285.112,A -85,B 0,C 180,E1 -6981.14,E2 -6981.14} C_VEL
LIN {X 0,Y 481.654,Z 285.119,A -85,B 0,C 180,E1 -6984.795,E2 -6984.795} C_VEL
LIN {X 0,Y 481.666,Z 285.114,A -85,B 0,C 180,E1 -6987.325,E2 -6987.325} C_VEL
LIN {X 0,Y 481.67,Z 285.113,A -85,B 0,C 180,E1 -6990.258,E2 -6990.258} C_VEL
LIN {X 0,Y 481.737,Z 285.103,A -85,B 0,C 180,E1 -6993.112,E2 -6993.112} C_VEL
LIN {X 0,Y 481.669,Z 285.112,A -85,B 0,C 180,E1 -6995.887,E2 -6995.887} C_VEL
LIN {X 0,Y 481.694,Z 285.108,A -85,B 0,C 180,E1 -6999.027,E2 -6999.027} C_VEL
LIN {X 0,Y 481.698,Z 285.106,A -85,B 0,C 180,E1 -7002.158,E2 -7002.158} C_VEL
LIN {X 0,Y 481.733,Z 285.105,A -85,B 0,C 180,E1 -7004.776,E2 -7004.776} C_VEL
LIN {X 0,Y 481.744,Z 285.101,A -85,B 0,C 180,E1 -7008.215,E2 -7008.215} C_VEL
LIN {X 0,Y 481.734,Z 285.101,A -85,B 0,C 180,E1 -7011.611,E2 -7011.611} C_VEL
LIN {X 0,Y 481.788,Z 285.096,A -85,B 0,C 180,E1 -7014.139,E2 -7014.139} C_VEL
LIN {X 0,Y 481.922,Z 285.077,A -85,B 0,C 180,E1 -7017.493,E2 -7017.493} C_VEL
LIN {X 0,Y 481.931,Z 285.082,A -85,B 0,C 180,E1 -7020,E2 -7020} C_VEL
LIN {X 0,Y 481.922,Z 285.079,A -85,B 0,C 180,E1 -7022.508,E2 -7022.508} C_VEL
LIN {X 0,Y 481.788,Z 285.098,A -85,B 0,C 180,E1 -7025.861,E2 -7025.861} C_VEL
LIN {X 0,Y 481.733,Z 285.1,A -85,B 0,C 180,E1 -7028.389,E2 -7028.389} C_VEL
LIN {X 0,Y 481.742,Z 285.1,A -85,B 0,C 180,E1 -7031.785,E2 -7031.785} C_VEL
LIN {X 0,Y 481.733,Z 285.105,A -85,B 0,C 180,E1 -7035.225,E2 -7035.225} C_VEL
LIN {X 0,Y 481.704,Z 285.108,A -85,B 0,C 180,E1 -7038.722,E2 -7038.722} C_VEL
LIN {X 0,Y 481.638,Z 285.118,A -85,B 0,C 180,E1 -7041.395,E2 -7041.395} C_VEL
LIN {X 0,Y 481.669,Z 285.112,A -85,B 0,C 180,E1 -7044.114,E2 -7044.114} C_VEL
LIN {X 0,Y 481.738,Z 285.102,A -85,B 0,C 180,E1 -7047.139,E2 -7047.139} C_VEL
LIN {X 0,Y 481.671,Z 285.108,A -85,B 0,C 180,E1 -7049.742,E2 -7049.742} C_VEL
LIN {X 0,Y 481.666,Z 285.109,A -85,B 0,C 180,E1 -7052.675,E2 -7052.675} C_VEL
LIN {X 0,Y 481.629,Z 285.115,A -85,B 0,C 180,E1 -7055.71,E2 -7055.71} C_VEL
LIN {X 0,Y 481.666,Z 285.112,A -85,B 0,C 180,E1 -7058.86,E2 -7058.86} C_VEL
LIN {X 0,Y 481.647,Z 285.115,A -85,B 0,C 180,E1 -7061.914,E2 -7061.914} C_VEL
LIN {X 0,Y 481.655,Z 285.117,A -85,B 0,C 180,E1 -7064.458,E2 -7064.458} C_VEL
LIN {X 0,Y 481.631,Z 285.119,A -85,B 0,C 180,E1 -7066.853,E2 -7066.853} C_VEL
LIN {X 0,Y 481.894,Z 288.366,A -85,B 0,C 180,E1 -7069.321,E2 -7069.321} C_VEL
LIN {X 0,Y 481.761,Z 292.399,A -85,B 0,C 180,E1 -7072.216,E2 -7072.216} C_VEL
LIN {X 0,Y 481.674,Z 296.871,A -85,B 0,C 180,E1 -7075.318,E2 -7075.318} C_VEL
LIN {X 0,Y 481.478,Z 301.334,A -85,B 0,C 180,E1 -7078.3,E2 -7078.3} C_VEL
LIN {X 0,Y 481.362,Z 305.784,A -85,B 0,C 180,E1 -7081.197,E2 -7081.197} C_VEL
LIN {X 0,Y 481.218,Z 310.261,A -85,B 0,C 180,E1 -7084.016,E2 -7084.016} C_VEL
LIN {X 0,Y 481.15,Z 315.055,A -85,B 0,C 180,E1 -7086.959,E2 -7086.959} C_VEL
LIN {X 0,Y 481.089,Z 316.023,A -85,B 0,C 180,E1 -7087.544,E2 -7087.544} C_VEL
LIN {X 0,Y 480.958,Z 317.455,A -85,B 0,C 180,E1 -7087.957,E2 -7087.957} C_VEL
LIN {X 0,Y 480.691,Z 319.884,A -85,B 0,C 180,E1 -7088.304,E2 -7088.304} C_VEL
LIN {X 0,Y 480.208,Z 324.651,A -85,B 0,C 180,E1 -7088.709,E2 -7088.709} C_VEL
LIN {X 0,Y 479.815,Z 330.351,A -85,B 0,C 180,E1 -7089.007,E2 -7089.007} C_VEL
LIN {X 0,Y 479.888,Z 338.453,A -85,B 0,C 180,E1 -7089.33,E2 -7089.33} C_VEL
LIN {X 0,Y 480.424,Z 342.452,A -85,B 0,C 180,E1 -7089.495,E2 -7089.495} C_VEL
LIN {X 0,Y 479.962,Z 357.298,A -85,B 0,C 180,E1 -7090.068,E2 -7090.068} C_VEL
LIN {X 0,Y 479.232,Z 370.587,A -85,B 0,C 180,E1 -7090.734,E2 -7090.734} C_VEL
LIN {X 0,Y 478.472,Z 384.205,A -85,B 0,C 180,E1 -7091.591,E2 -7091.591} C_VEL
LIN {X 0,Y 477.704,Z 396.729,A -85,B 0,C 180,E1 -7092.558,E2 -7092.558} C_VEL
LIN {X 0,Y 476.906,Z 409.414,A -85,B 0,C 180,E1 -7093.741,E2 -7093.741} C_VEL
LIN {X 0,Y 476.152,Z 420.917,A -85,B 0,C 180,E1 -7095.031,E2 -7095.031} C_VEL
LIN {X 0,Y 475.506,Z 430.598,A -85,B 0,C 180,E1 -7096.322,E2 -7096.322} C_VEL
LIN {X 0,Y 474.94,Z 439.676,A -85,B 0,C 180,E1 -7097.754,E2 -7097.754} C_VEL
LIN {X 0,Y 474.535,Z 447.991,A -85,B 0,C 180,E1 -7099.332,E2 -7099.332} C_VEL
LIN {X 0,Y 474.146,Z 455.371,A -85,B 0,C 180,E1 -7101.047,E2 -7101.047} C_VEL
LIN {X 0,Y 473.922,Z 461.229,A -85,B 0,C 180,E1 -7102.759,E2 -7102.759} C_VEL
LIN {X 0,Y 473.87,Z 464.698,A -85,B 0,C 180,E1 -7104.041,E2 -7104.041} C_VEL
LIN {X 0,Y 473.711,Z 468.217,A -85,B 0,C 180,E1 -7105.746,E2 -7105.746} C_VEL
LIN {X 0,Y 473.737,Z 470.545,A -85,B 0,C 180,E1 -7107.45,E2 -7107.45} C_VEL
LIN {X 0,Y 473.685,Z 471.737,A -85,B 0,C 180,E1 -7109.15,E2 -7109.15} C_VEL
LIN {X 0,Y 473.686,Z 471.755,A -85,B 0,C 180,E1 -7110.85,E2 -7110.85} C_VEL
LIN {X 0,Y 473.737,Z 470.633,A -85,B 0,C 180,E1 -7112.551,E2 -7112.551} C_VEL
LIN {X 0,Y 473.71,Z 468.373,A -85,B 0,C 180,E1 -7114.254,E2 -7114.254} C_VEL
LIN {X 0,Y 473.841,Z 464.919,A -85,B 0,C 180,E1 -7115.96,E2 -7115.96} C_VEL
LIN {X 0,Y 473.975,Z 460.191,A -85,B 0,C 180,E1 -7117.669,E2 -7117.669} C_VEL
LIN {X 0,Y 474.209,Z 454.066,A -85,B 0,C 180,E1 -7119.383,E2 -7119.383} C_VEL
LIN {X 0,Y 474.652,Z 446.354,A -85,B 0,C 180,E1 -7121.098,E2 -7121.098} C_VEL
LIN {X 0,Y 475.042,Z 438.041,A -85,B 0,C 180,E1 -7122.62,E2 -7122.62} C_VEL
LIN {X 0,Y 475.672,Z 428.235,A -85,B 0,C 180,E1 -7124.11,E2 -7124.11} C_VEL
LIN {X 0,Y 476.286,Z 418.086,A -85,B 0,C 180,E1 -7125.403,E2 -7125.403} C_VEL
LIN {X 0,Y 477.032,Z 407.155,A -85,B 0,C 180,E1 -7126.577,E2 -7126.577} C_VEL
LIN {X 0,Y 477.804,Z 395.189,A -85,B 0,C 180,E1 -7127.66,E2 -7127.66} C_VEL
LIN {X 0,Y 478.585,Z 382.327,A -85,B 0,C 180,E1 -7128.627,E2 -7128.627} C_VEL
LIN {X 0,Y 479.291,Z 370.21,A -85,B 0,C 180,E1 -7129.376,E2 -7129.376} C_VEL
LIN {X 0,Y 479.941,Z 356.195,A -85,B 0,C 180,E1 -7130.071,E2 -7130.071} C_VEL
LIN {X 0,Y 480.303,Z 341.998,A -85,B 0,C 180,E1 -7130.616,E2 -7130.616} C_VEL
LIN {X 0,Y 476.691,Z 327.865,A -85,B 0,C 180,E1 -7131.177,E2 -7131.177} C_VEL
LIN {X 0,Y 473.98,Z 318.391,A -85,B 0,C 180,E1 -7131.503,E2 -7131.503} C_VEL
LIN {X 0,Y 474.11,Z 313.508,A -85,B 0,C 180,E1 -7134.523,E2 -7134.523} C_VEL
LIN {X 0,Y 474.215,Z 309.047,A -85,B 0,C 180,E1 -7137.35,E2 -7137.35} C_VEL
LIN {X 0,Y 474.37,Z 304.565,A -85,B 0,C 180,E1 -7140.247,E2 -7140.247} C_VEL
LIN {X 0,Y 474.501,Z 300.076,A -85,B 0,C 180,E1 -7143.231,E2 -7143.231} C_VEL
LIN {X 0,Y 474.665,Z 295.578,A -85,B 0,C 180,E1 -7146.316,E2 -7146.316} C_VEL
LIN {X 0,Y 474.846,Z 290.867,A -85,B 0,C 180,E1 -7149.679,E2 -7149.679} C_VEL
LIN {X 0,Y 474.777,Z 287.429,A -85,B 0,C 180,E1 -7152.257,E2 -7152.257} C_VEL
LIN {X 0,Y 474.601,Z 285.994,A -85,B 0,C 180,E1 -7153.481,E2 -7153.481} C_VEL
LIN {X 0,Y 474.6,Z 285.994,A -85,B 0,C 180,E1 -7156.519,E2 -7156.519} C_VEL
LIN {X 0,Y 474.615,Z 285.989,A -85,B 0,C 180,E1 -7159.342,E2 -7159.342} C_VEL
LIN {X 0,Y 474.608,Z 285.995,A -85,B 0,C 180,E1 -7161.704,E2 -7161.704} C_VEL
LIN {X 0,Y 474.621,Z 285.993,A -85,B 0,C 180,E1 -7164.725,E2 -7164.725} C_VEL
LIN {X 0,Y 474.633,Z 285.991,A -85,B 0,C 180,E1 -7167.787,E2 -7167.787} C_VEL
LIN {X 0,Y 474.604,Z 285.995,A -85,B 0,C 180,E1 -7170.888,E2 -7170.888} C_VEL
LIN {X 0,Y 474.612,Z 285.989,A -85,B 0,C 180,E1 -7173.625,E2 -7173.625} C_VEL
LIN {X 0,Y 474.632,Z 285.988,A -85,B 0,C 180,E1 -7176.641,E2 -7176.641} C_VEL
LIN {X 0,Y 474.651,Z 285.988,A -85,B 0,C 180,E1 -7180.089,E2 -7180.089} C_VEL
LIN {X 0,Y 474.647,Z 285.986,A -85,B 0,C 180,E1 -7182.774,E2 -7182.774} C_VEL
LIN {X 0,Y 474.639,Z 285.986,A -85,B 0,C 180,E1 -7185.421,E2 -7185.421} C_VEL
LIN {X 0,Y 474.701,Z 285.981,A -85,B 0,C 180,E1 -7188.037,E2 -7188.037} C_VEL
LIN {X 0,Y 474.71,Z 285.977,A -85,B 0,C 180,E1 -7191.486,E2 -7191.486} C_VEL
LIN {X 0,Y 474.744,Z 285.973,A -85,B 0,C 180,E1 -7194.904,E2 -7194.904} C_VEL
LIN {X 0,Y 474.892,Z 285.955,A -85,B 0,C 180,E1 -7197.455,E2 -7197.455} C_VEL
LIN {X 0,Y 474.905,Z 285.957,A -85,B 0,C 180,E1 -7200,E2 -7200} C_VEL
LIN {X 0,Y 474.892,Z 285.955,A -85,B 0,C 180,E1 -7202.545,E2 -7202.545} C_VEL
LIN {X 0,Y 474.753,Z 285.974,A -85,B 0,C 180,E1 -7205.948,E2 -7205.948} C_VEL
LIN {X 0,Y 474.71,Z 285.977,A -85,B 0,C 180,E1 -7208.514,E2 -7208.514} C_VEL
LIN {X 0,Y 474.701,Z 285.981,A -85,B 0,C 180,E1 -7211.962,E2 -7211.962} C_VEL
LIN {X 0,Y 474.696,Z 285.983,A -85,B 0,C 180,E1 -7215.456,E2 -7215.456} C_VEL
LIN {X 0,Y 474.661,Z 285.983,A -85,B 0,C 180,E1 -7219.01,E2 -7219.01} C_VEL
LIN {X 0,Y 474.584,Z 285.995,A -85,B 0,C 180,E1 -7221.729,E2 -7221.729} C_VEL
LIN {X 0,Y 474.652,Z 285.989,A -85,B 0,C 180,E1 -7224.493,E2 -7224.493} C_VEL
LIN {X 0,Y 474.676,Z 285.985,A -85,B 0,C 180,E1 -7227.334,E2 -7227.334} C_VEL
LIN {X 0,Y 474.6,Z 285.997,A -85,B 0,C 180,E1 -7230.81,E2 -7230.81} C_VEL
LIN {X 0,Y 474.634,Z 285.993,A -85,B 0,C 180,E1 -7233.984,E2 -7233.984} C_VEL
LIN {X 0,Y 474.568,Z 286.002,A -85,B 0,C 180,E1 -7236.899,E2 -7236.899} C_VEL
LIN {X 0,Y 474.611,Z 285.995,A -85,B 0,C 180,E1 -7239.646,E2 -7239.646} C_VEL
LIN {X 0,Y 474.598,Z 285.993,A -85,B 0,C 180,E1 -7242.234,E2 -7242.234} C_VEL
LIN {X 0,Y 474.649,Z 286.012,A -85,B 0,C 180,E1 -7245.294,E2 -7245.294} C_VEL
LIN {X 0,Y 475.128,Z 289.541,A -85,B 0,C 180,E1 -7247.696,E2 -7247.696} C_VEL
LIN {X 0,Y 475.216,Z 292.188,A -85,B 0,C 180,E1 -7249.405,E2 -7249.405} C_VEL
LIN {X 0,Y 474.996,Z 297.479,A -85,B 0,C 180,E1 -7252.654,E2 -7252.654} C_VEL
LIN {X 0,Y 474.874,Z 301.004,A -85,B 0,C 180,E1 -7254.747,E2 -7254.747} C_VEL
LIN {X 0,Y 474.679,Z 306.296,A -85,B 0,C 180,E1 -7257.791,E2 -7257.791} C_VEL
LIN {X 0,Y 474.456,Z 311.936,A -85,B 0,C 180,E1 -7260.921,E2 -7260.921} C_VEL
LIN {X 0,Y 474.265,Z 316.927,A -85,B 0,C 180,E1 -7263.605,E2 -7263.605} C_VEL
LIN {X 0,Y 474.132,Z 322.967,A -85,B 0,C 180,E1 -7266.783,E2 -7266.783} C_VEL
LIN {X 0,Y 474.038,Z 326.375,A -85,B 0,C 180,E1 -7268.54,E2 -7268.54} C_VEL
LIN {X 0,Y 478.672,Z 343.978,A -85,B 0,C 180,E1 -7269.148,E2 -7269.148} C_VEL
LIN {X 0,Y 480.355,Z 351.769,A -85,B 0,C 180,E1 -7269.468,E2 -7269.468} C_VEL
LIN {X 0,Y 479.852,Z 366.518,A -85,B 0,C 180,E1 -7270.04,E2 -7270.04} C_VEL
LIN {X 0,Y 479.081,Z 380.187,A -85,B 0,C 180,E1 -7270.727,E2 -7270.727} C_VEL
LIN {X 0,Y 478.302,Z 393.67,A -85,B 0,C 180,E1 -7271.584,E2 -7271.584} C_VEL
LIN {X 0,Y 477.497,Z 407.393,A -85,B 0,C 180,E1 -7272.66,E2 -7272.66} C_VEL
LIN {X 0,Y 476.721,Z 419.812,A -85,B 0,C 180,E1 -7273.843,E2 -7273.843} C_VEL
LIN {X 0,Y 476.008,Z 430.221,A -85,B 0,C 180,E1 -7275.026,E2 -7275.026} C_VEL
LIN {X 0,Y 475.398,Z 439.882,A -85,B 0,C 180,E1 -7276.318,E2 -7276.318} C_VEL
LIN {X 0,Y 474.807,Z 449.393,A -85,B 0,C 180,E1 -7277.828,E2 -7277.828} C_VEL
LIN {X 0,Y 474.483,Z 457.271,A -85,B 0,C 180,E1 -7279.33,E2 -7279.33} C_VEL
LIN {X 0,Y 474.095,Z 464.646,A -85,B 0,C 180,E1 -7281.045,E2 -7281.045} C_VEL
LIN {X 0,Y 473.909,Z 470.495,A -85,B 0,C 180,E1 -7282.758,E2 -7282.758} C_VEL
LIN {X 0,Y 473.812,Z 473.971,A -85,B 0,C 180,E1 -7284.04,E2 -7284.04} C_VEL
LIN {X 0,Y 473.703,Z 477.483,A -85,B 0,C 180,E1 -7285.746,E2 -7285.746} C_VEL
LIN {X 0,Y 473.718,Z 479.794,A -85,B 0,C 180,E1 -7287.449,E2 -7287.449} C_VEL
LIN {X 0,Y 473.684,Z 480.957,A -85,B 0,C 180,E1 -7289.15,E2 -7289.15} C_VEL
LIN {X 0,Y 473.684,Z 480.956,A -85,B 0,C 180,E1 -7290.85,E2 -7290.85} C_VEL
LIN {X 0,Y 473.718,Z 479.791,A -85,B 0,C 180,E1 -7292.551,E2 -7292.551} C_VEL
LIN {X 0,Y 473.703,Z 477.48,A -85,B 0,C 180,E1 -7294.254,E2 -7294.254} C_VEL
LIN {X 0,Y 473.833,Z 473.974,A -85,B 0,C 180,E1 -7295.959,E2 -7295.959} C_VEL
LIN {X 0,Y 473.943,Z 469.182,A -85,B 0,C 180,E1 -7297.669,E2 -7297.669} C_VEL
LIN {X 0,Y 474.171,Z 462.974,A -85,B 0,C 180,E1 -7299.383,E2 -7299.383} C_VEL
LIN {X 0,Y 474.599,Z 455.176,A -85,B 0,C 180,E1 -7301.099,E2 -7301.099} C_VEL
LIN {X 0,Y 474.947,Z 447.456,A -85,B 0,C 180,E1 -7302.509,E2 -7302.509} C_VEL
LIN {X 0,Y 475.616,Z 436.884,A -85,B 0,C 180,E1 -7304.111,E2 -7304.111} C_VEL
LIN {X 0,Y 476.221,Z 426.656,A -85,B 0,C 180,E1 -7305.404,E2 -7305.404} C_VEL
LIN {X 0,Y 477.058,Z 413.912,A -85,B 0,C 180,E1 -7306.749,E2 -7306.749} C_VEL
LIN {X 0,Y 477.881,Z 400.903,A -85,B 0,C 180,E1 -7307.878,E2 -7307.878} C_VEL
LIN {X 0,Y 478.692,Z 387.297,A -85,B 0,C 180,E1 -7308.844,E2 -7308.844} C_VEL
LIN {X 0,Y 479.477,Z 373.203,A -85,B 0,C 180,E1 -7309.645,E2 -7309.645} C_VEL
LIN {X 0,Y 480.118,Z 357.754,A -85,B 0,C 180,E1 -7310.324,E2 -7310.324} C_VEL
LIN {X 0,Y 480.182,Z 350.691,A -85,B 0,C 180,E1 -7310.578,E2 -7310.578} C_VEL
LIN {X 0,Y 476.437,Z 335.259,A -85,B 0,C 180,E1 -7311.173,E2 -7311.173} C_VEL
LIN {X 0,Y 474.021,Z 326.398,A -85,B 0,C 180,E1 -7311.457,E2 -7311.457} C_VEL
LIN {X 0,Y 474.162,Z 320.519,A -85,B 0,C 180,E1 -7314.519,E2 -7314.519} C_VEL
LIN {X 0,Y 474.324,Z 315.222,A -85,B 0,C 180,E1 -7317.343,E2 -7317.343} C_VEL
LIN {X 0,Y 474.515,Z 309.894,A -85,B 0,C 180,E1 -7320.236,E2 -7320.236} C_VEL
LIN {X 0,Y 474.72,Z 304.56,A -85,B 0,C 180,E1 -7323.213,E2 -7323.213} C_VEL
LIN {X 0,Y 474.941,Z 299.241,A -85,B 0,C 180,E1 -7326.291,E2 -7326.291} C_VEL
LIN {X 0,Y 475.143,Z 293.937,A -85,B 0,C 180,E1 -7329.495,E2 -7329.495} C_VEL
LIN {X 0,Y 475.17,Z 290.404,A -85,B 0,C 180,E1 -7331.725,E2 -7331.725} C_VEL
LIN {X 0,Y 474.794,Z 286.886,A -85,B 0,C 180,E1 -7334.082,E2 -7334.082} C_VEL
LIN {X 0,Y 474.631,Z 285.991,A -85,B 0,C 180,E1 -7334.871,E2 -7334.871} C_VEL
LIN {X 0,Y 474.614,Z 285.993,A -85,B 0,C 180,E1 -7338.214,E2 -7338.214} C_VEL
LIN {X 0,Y 474.638,Z 285.99,A -85,B 0,C 180,E1 -7340.454,E2 -7340.454} C_VEL
LIN {X 0,Y 474.581,Z 285.997,A -85,B 0,C 180,E1 -7343.676,E2 -7343.676} C_VEL
LIN {X 0,Y 474.636,Z 285.991,A -85,B 0,C 180,E1 -7346.779,E2 -7346.779} C_VEL
LIN {X 0,Y 474.598,Z 285.995,A -85,B 0,C 180,E1 -7349.769,E2 -7349.769} C_VEL
LIN {X 0,Y 474.689,Z 285.984,A -85,B 0,C 180,E1 -7352.679,E2 -7352.679} C_VEL
LIN {X 0,Y 474.651,Z 285.99,A -85,B 0,C 180,E1 -7355.507,E2 -7355.507} C_VEL
LIN {X 0,Y 474.662,Z 285.984,A -85,B 0,C 180,E1 -7359.185,E2 -7359.185} C_VEL
LIN {X 0,Y 474.648,Z 285.986,A -85,B 0,C 180,E1 -7361.884,E2 -7361.884} C_VEL
LIN {X 0,Y 474.691,Z 285.983,A -85,B 0,C 180,E1 -7364.544,E2 -7364.544} C_VEL
LIN {X 0,Y 474.697,Z 285.98,A -85,B 0,C 180,E1 -7368.037,E2 -7368.037} C_VEL
LIN {X 0,Y 474.705,Z 285.977,A -85,B 0,C 180,E1 -7371.486,E2 -7371.486} C_VEL
LIN {X 0,Y 474.741,Z 285.972,A -85,B 0,C 180,E1 -7374.904,E2 -7374.904} C_VEL
LIN {X 0,Y 474.888,Z 285.953,A -85,B 0,C 180,E1 -7377.455,E2 -7377.455} C_VEL
LIN {X 0,Y 474.901,Z 285.958,A -85,B 0,C 180,E1 -7380,E2 -7380} C_VEL
LIN {X 0,Y 474.888,Z 285.955,A -85,B 0,C 180,E1 -7382.545,E2 -7382.545} C_VEL
LIN {X 0,Y 474.749,Z 285.975,A -85,B 0,C 180,E1 -7385.948,E2 -7385.948} C_VEL
LIN {X 0,Y 474.705,Z 285.975,A -85,B 0,C 180,E1 -7388.514,E2 -7388.514} C_VEL
LIN {X 0,Y 474.696,Z 285.979,A -85,B 0,C 180,E1 -7391.963,E2 -7391.963} C_VEL
LIN {X 0,Y 474.691,Z 285.983,A -85,B 0,C 180,E1 -7395.456,E2 -7395.456} C_VEL
LIN {X 0,Y 474.657,Z 285.984,A -85,B 0,C 180,E1 -7399.011,E2 -7399.011} C_VEL
LIN {X 0,Y 474.581,Z 285.995,A -85,B 0,C 180,E1 -7401.729,E2 -7401.729} C_VEL
LIN {X 0,Y 474.651,Z 285.988,A -85,B 0,C 180,E1 -7404.493,E2 -7404.493} C_VEL
LIN {X 0,Y 474.672,Z 285.984,A -85,B 0,C 180,E1 -7407.335,E2 -7407.335} C_VEL
LIN {X 0,Y 474.598,Z 285.992,A -85,B 0,C 180,E1 -7410.811,E2 -7410.811} C_VEL
LIN {X 0,Y 474.63,Z 285.987,A -85,B 0,C 180,E1 -7413.984,E2 -7413.984} C_VEL
LIN {X 0,Y 474.565,Z 285.998,A -85,B 0,C 180,E1 -7416.9,E2 -7416.9} C_VEL
LIN {X 0,Y 474.622,Z 285.992,A -85,B 0,C 180,E1 -7419.648,E2 -7419.648} C_VEL
LIN {X 0,Y 474.609,Z 285.994,A -85,B 0,C 180,E1 -7422.935,E2 -7422.935} C_VEL
LIN {X 0,Y 474.603,Z 285.995,A -85,B 0,C 180,E1 -7425.896,E2 -7425.896} C_VEL
LIN {X 0,Y 474.592,Z 285.996,A -85,B 0,C 180,E1 -7426.52,E2 -7426.52} C_VEL
LIN {X 0,Y 474.785,Z 287.953,A -85,B 0,C 180,E1 -7428.234,E2 -7428.234} C_VEL
LIN {X 0,Y 474.815,Z 290.941,A -85,B 0,C 180,E1 -7430.472,E2 -7430.472} C_VEL
LIN {X 0,Y 474.662,Z 295.424,A -85,B 0,C 180,E1 -7433.684,E2 -7433.684} C_VEL
LIN {X 0,Y 474.498,Z 299.895,A -85,B 0,C 180,E1 -7436.769,E2 -7436.769} C_VEL
LIN {X 0,Y 474.372,Z 304.355,A -85,B 0,C 180,E1 -7439.754,E2 -7439.754} C_VEL
LIN {X 0,Y 474.211,Z 309.018,A -85,B 0,C 180,E1 -7442.776,E2 -7442.776} C_VEL
LIN {X 0,Y 474.11,Z 313.313,A -85,B 0,C 180,E1 -7445.478,E2 -7445.478} C_VEL
LIN {X 0,Y 473.985,Z 318.392,A -85,B 0,C 180,E1 -7448.602,E2 -7448.602} C_VEL
LIN {X 0,Y 478.558,Z 334.564,A -85,B 0,C 180,E1 -7449.167,E2 -7449.167} C_VEL
LIN {X 0,Y 480.424,Z 342.452,A -85,B 0,C 180,E1 -7449.495,E2 -7449.495} C_VEL
LIN {X 0,Y 480.544,Z 346.134,A -85,B 0,C 180,E1 -7449.633,E2 -7449.633} C_VEL
LIN {X 0,Y 479.837,Z 349.855,A -85,B 0,C 180,E1 -7449.742,E2 -7449.742} C_VEL
LIN {X 0,Y 477.201,Z 357.163,A -85,B 0,C 180,E1 -7449.94,E2 -7449.94} C_VEL
LIN {X 0,Y 473.522,Z 366.252,A -85,B 0,C 180,E1 -7450.239,E2 -7450.239} C_VEL
LIN {X 0,Y 472.462,Z 371.728,A -85,B 0,C 180,E1 -7450.51,E2 -7450.51} C_VEL
LIN {X 0,Y 471.625,Z 385.846,A -85,B 0,C 180,E1 -7451.427,E2 -7451.427} C_VEL
LIN {X 0,Y 470.771,Z 399.352,A -85,B 0,C 180,E1 -7452.517,E2 -7452.517} C_VEL
LIN {X 0,Y 469.895,Z 411.603,A -85,B 0,C 180,E1 -7453.714,E2 -7453.714} C_VEL
LIN {X 0,Y 469.108,Z 422.765,A -85,B 0,C 180,E1 -7455.023,E2 -7455.023} C_VEL
LIN {X 0,Y 468.35,Z 433.611,A -85,B 0,C 180,E1 -7456.551,E2 -7456.551} C_VEL
LIN {X 0,Y 467.814,Z 442.611,A -85,B 0,C 180,E1 -7458.079,E2 -7458.079} C_VEL
LIN {X 0,Y 467.345,Z 450.073,A -85,B 0,C 180,E1 -7459.604,E2 -7459.604} C_VEL
LIN {X 0,Y 467.043,Z 457.051,A -85,B 0,C 180,E1 -7461.346,E2 -7461.346} C_VEL
LIN {X 0,Y 466.83,Z 462.537,A -85,B 0,C 180,E1 -7463.083,E2 -7463.083} C_VEL
LIN {X 0,Y 466.732,Z 466.681,A -85,B 0,C 180,E1 -7464.817,E2 -7464.817} C_VEL
LIN {X 0,Y 466.674,Z 469.595,A -85,B 0,C 180,E1 -7466.547,E2 -7466.547} C_VEL
LIN {X 0,Y 466.605,Z 471.351,A -85,B 0,C 180,E1 -7468.274,E2 -7468.274} C_VEL
LIN {X 0,Y 466.597,Z 471.965,A -85,B 0,C 180,E1 -7470,E2 -7470} C_VEL
LIN {X 0,Y 466.605,Z 471.403,A -85,B 0,C 180,E1 -7471.727,E2 -7471.727} C_VEL
LIN {X 0,Y 466.675,Z 469.716,A -85,B 0,C 180,E1 -7473.454,E2 -7473.454} C_VEL
LIN {X 0,Y 466.725,Z 466.867,A -85,B 0,C 180,E1 -7475.184,E2 -7475.184} C_VEL
LIN {X 0,Y 466.823,Z 462.788,A -85,B 0,C 180,E1 -7476.918,E2 -7476.918} C_VEL
LIN {X 0,Y 467.033,Z 457.38,A -85,B 0,C 180,E1 -7478.655,E2 -7478.655} C_VEL
LIN {X 0,Y 467.328,Z 450.49,A -85,B 0,C 180,E1 -7480.397,E2 -7480.397} C_VEL
LIN {X 0,Y 467.779,Z 443.081,A -85,B 0,C 180,E1 -7481.922,E2 -7481.922} C_VEL
LIN {X 0,Y 468.307,Z 434.158,A -85,B 0,C 180,E1 -7483.451,E2 -7483.451} C_VEL
LIN {X 0,Y 468.933,Z 425.063,A -85,B 0,C 180,E1 -7484.761,E2 -7484.761} C_VEL
LIN {X 0,Y 469.676,Z 414.335,A -85,B 0,C 180,E1 -7486.071,E2 -7486.071} C_VEL
LIN {X 0,Y 470.494,Z 403.105,A -85,B 0,C 180,E1 -7487.225,E2 -7487.225} C_VEL
LIN {X 0,Y 471.378,Z 389.843,A -85,B 0,C 180,E1 -7488.359,E2 -7488.359} C_VEL
LIN {X 0,Y 472.217,Z 375.74,A -85,B 0,C 180,E1 -7489.338,E2 -7489.338} C_VEL
LIN {X 0,Y 473.097,Z 360.926,A -85,B 0,C 180,E1 -7490.147,E2 -7490.147} C_VEL
LIN {X 0,Y 473.681,Z 346.605,A -85,B 0,C 180,E1 -7490.749,E2 -7490.749} C_VEL
LIN {X 0,Y 473.551,Z 342.87,A -85,B 0,C 180,E1 -7490.895,E2 -7490.895} C_VEL
LIN {X 0,Y 469.841,Z 328.461,A -85,B 0,C 180,E1 -7491.487,E2 -7491.487} C_VEL
LIN {X 0,Y 466.927,Z 318.456,A -85,B 0,C 180,E1 -7491.847,E2 -7491.847} C_VEL
LIN {X 0,Y 467.068,Z 313.574,A -85,B 0,C 180,E1 -7494.918,E2 -7494.918} C_VEL
LIN {X 0,Y 467.169,Z 309.097,A -85,B 0,C 180,E1 -7497.798,E2 -7497.798} C_VEL
LIN {X 0,Y 467.364,Z 304.62,A -85,B 0,C 180,E1 -7500.749,E2 -7500.749} C_VEL
LIN {X 0,Y 467.557,Z 299.483,A -85,B 0,C 180,E1 -7504.236,E2 -7504.236} C_VEL
LIN {X 0,Y 467.654,Z 295.266,A -85,B 0,C 180,E1 -7507.203,E2 -7507.203} C_VEL
LIN {X 0,Y 467.835,Z 291.108,A -85,B 0,C 180,E1 -7510.238,E2 -7510.238} C_VEL
LIN {X 0,Y 467.694,Z 288.069,A -85,B 0,C 180,E1 -7512.581,E2 -7512.581} C_VEL
LIN {X 0,Y 467.553,Z 286.873,A -85,B 0,C 180,E1 -7513.821,E2 -7513.821} C_VEL
LIN {X 0,Y 467.555,Z 286.872,A -85,B 0,C 180,E1 -7516.255,E2 -7516.255} C_VEL
LIN {X 0,Y 467.577,Z 286.87,A -85,B 0,C 180,E1 -7518.723,E2 -7518.723} C_VEL
LIN {X 0,Y 467.563,Z 286.872,A -85,B 0,C 180,E1 -7521.955,E2 -7521.955} C_VEL
LIN {X 0,Y 467.561,Z 286.871,A -85,B 0,C 180,E1 -7525.167,E2 -7525.167} C_VEL
LIN {X 0,Y 467.58,Z 286.868,A -85,B 0,C 180,E1 -7528.26,E2 -7528.26} C_VEL
LIN {X 0,Y 467.553,Z 286.871,A -85,B 0,C 180,E1 -7531.249,E2 -7531.249} C_VEL
LIN {X 0,Y 467.581,Z 286.869,A -85,B 0,C 180,E1 -7534.158,E2 -7534.158} C_VEL
LIN {X 0,Y 467.573,Z 286.87,A -85,B 0,C 180,E1 -7536.996,E2 -7536.996} C_VEL
LIN {X 0,Y 467.619,Z 286.862,A -85,B 0,C 180,E1 -7539.777,E2 -7539.777} C_VEL
LIN {X 0,Y 467.605,Z 286.862,A -85,B 0,C 180,E1 -7542.507,E2 -7542.507} C_VEL
LIN {X 0,Y 467.599,Z 286.864,A -85,B 0,C 180,E1 -7545.196,E2 -7545.196} C_VEL
LIN {X 0,Y 467.653,Z 286.859,A -85,B 0,C 180,E1 -7547.854,E2 -7547.854} C_VEL
LIN {X 0,Y 467.668,Z 286.854,A -85,B 0,C 180,E1 -7551.357,E2 -7551.357} C_VEL
LIN {X 0,Y 467.715,Z 286.853,A -85,B 0,C 180,E1 -7553.962,E2 -7553.962} C_VEL
LIN {X 0,Y 467.857,Z 286.831,A -85,B 0,C 180,E1 -7557.417,E2 -7557.417} C_VEL
LIN {X 0,Y 467.875,Z 286.832,A -85,B 0,C 180,E1 -7560,E2 -7560} C_VEL
LIN {X 0,Y 467.857,Z 286.831,A -85,B 0,C 180,E1 -7562.583,E2 -7562.583} C_VEL
LIN {X 0,Y 467.715,Z 286.852,A -85,B 0,C 180,E1 -7566.038,E2 -7566.038} C_VEL
LIN {X 0,Y 467.661,Z 286.857,A -85,B 0,C 180,E1 -7569.515,E2 -7569.515} C_VEL
LIN {X 0,Y 467.65,Z 286.861,A -85,B 0,C 180,E1 -7572.358,E2 -7572.358} C_VEL
LIN {X 0,Y 467.646,Z 286.858,A -85,B 0,C 180,E1 -7575.885,E2 -7575.885} C_VEL
LIN {X 0,Y 467.619,Z 286.861,A -85,B 0,C 180,E1 -7579.308,E2 -7579.308} C_VEL
